   DATA[2489,28] := 261.6637;
   DATA[2489,29] := 12.11228;
   DATA[2489,30] := 1.723661;
   DATA[2489,31] := 1.271551;
   DATA[2489,32] := 0.7353967;
   DATA[2489,33] := 0.3084905;
   DATA[2489,34] := 2.0;
   DATA[2489,35] := 249.9199;
   DATA[2489,36] := 1.681991;
   DATA[2489,37] := 188.7817;
   DATA[2489,38] := 0.000128152;
   DATA[2489,39] := 1.0;
   DATA[2489,40] := 1.0;
   DATA[2490,0] := 2.585274;
   DATA[2490,1] := 868.7028;
   DATA[2490,2] := 2.0;
   DATA[2490,3] := 2.0;
   DATA[2490,4] := 262.3045;
   DATA[2490,5] := 8.396437;
   DATA[2490,6] := 329.7103;
   DATA[2490,7] := 2.455131;
   DATA[2490,8] := 2.0;
   DATA[2490,9] := 2.0;
   DATA[2490,10] := 2.0;
   DATA[2490,11] := 19.80601;
   DATA[2490,12] := 2.208884;
   DATA[2490,13] := 824.428;
   DATA[2490,14] := 1.0;
   DATA[2490,15] := 2.0;
   DATA[2490,16] := 1.0;
   DATA[2490,17] := 1.0;
   DATA[2490,18] := 1.0;
   DATA[2490,19] := 2.0;
   DATA[2490,20] := 148.808;
   DATA[2490,21] := 155.2166;
   DATA[2490,22] := 1.714798;
   DATA[2490,23] := 867.4699;
   DATA[2490,24] := 2.0;
   DATA[2490,25] := 2.0;
   DATA[2490,26] := 7.874135;
   DATA[2490,27] := 144.9628;
   DATA[2490,28] := 261.6637;
   DATA[2490,29] := 11.95847;
   DATA[2490,30] := 1.723661;
   DATA[2490,31] := 1.257333;
   DATA[2490,32] := 0.7353967;
   DATA[2490,33] := 0.3084905;
   DATA[2490,34] := 2.0;
   DATA[2490,35] := 249.9199;
   DATA[2490,36] := 1.681991;
   DATA[2490,37] := 188.7817;
   DATA[2490,38] := 0.000128152;
   DATA[2490,39] := 1.0;
   DATA[2490,40] := 1.0;
   DATA[2491,0] := 2.562854;
   DATA[2491,1] := 868.6635;
   DATA[2491,2] := 2.0;
   DATA[2491,3] := 2.0;
   DATA[2491,4] := 262.4007;
   DATA[2491,5] := 8.396437;
   DATA[2491,6] := 329.7103;
   DATA[2491,7] := 2.4559;
   DATA[2491,8] := 2.0;
   DATA[2491,9] := 2.0;
   DATA[2491,10] := 2.0;
   DATA[2491,11] := 19.77079;
   DATA[2491,12] := 2.208884;
   DATA[2491,13] := 825.0289;
   DATA[2491,14] := 1.0;
   DATA[2491,15] := 2.0;
   DATA[2491,16] := 1.0;
   DATA[2491,17] := 1.0;
   DATA[2491,18] := 1.0;
   DATA[2491,19] := 2.0;
   DATA[2491,20] := 148.808;
   DATA[2491,21] := 155.2166;
   DATA[2491,22] := 1.71608;
   DATA[2491,23] := 867.5468;
   DATA[2491,24] := 2.0;
   DATA[2491,25] := 2.0;
   DATA[2491,26] := 7.874135;
   DATA[2491,27] := 144.9628;
   DATA[2491,28] := 261.5355;
   DATA[2491,29] := 11.95847;
   DATA[2491,30] := 1.72507;
   DATA[2491,31] := 1.256565;
   DATA[2491,32] := 0.7353967;
   DATA[2491,33] := 0.3084905;
   DATA[2491,34] := 2.0;
   DATA[2491,35] := 249.9199;
   DATA[2491,36] := 1.681991;
   DATA[2491,37] := 188.7817;
   DATA[2491,38] := 0.000128152;
   DATA[2491,39] := 1.0;
   DATA[2491,40] := 1.0;
   DATA[2492,0] := 2.540115;
   DATA[2492,1] := 869.0953;
   DATA[2492,2] := 2.0;
   DATA[2492,3] := 2.0;
   DATA[2492,4] := 262.4007;
   DATA[2492,5] := 8.396437;
   DATA[2492,6] := 329.6591;
   DATA[2492,7] := 2.4559;
   DATA[2492,8] := 2.0;
   DATA[2492,9] := 2.0;
   DATA[2492,10] := 2.0;
   DATA[2492,11] := 19.72598;
   DATA[2492,12] := 2.208884;
   DATA[2492,13] := 825.0689;
   DATA[2492,14] := 1.0;
   DATA[2492,15] := 2.0;
   DATA[2492,16] := 1.0;
   DATA[2492,17] := 1.0;
   DATA[2492,18] := 1.0;
   DATA[2492,19] := 2.0;
   DATA[2492,20] := 148.808;
   DATA[2492,21] := 155.2166;
   DATA[2492,22] := 1.71608;
   DATA[2492,23] := 867.739;
   DATA[2492,24] := 2.0;
   DATA[2492,25] := 2.0;
   DATA[2492,26] := 7.874135;
   DATA[2492,27] := 144.9628;
   DATA[2492,28] := 261.5034;
   DATA[2492,29] := 11.95847;
   DATA[2492,30] := 1.72507;
   DATA[2492,31] := 1.261176;
   DATA[2492,32] := 0.7353967;
   DATA[2492,33] := 0.3084905;
   DATA[2492,34] := 2.0;
   DATA[2492,35] := 249.9199;
   DATA[2492,36] := 1.649953;
   DATA[2492,37] := 188.7817;
   DATA[2492,38] := 0.000128152;
   DATA[2492,39] := 1.0;
   DATA[2492,40] := 1.0;
   DATA[2493,0] := 2.524421;
   DATA[2493,1] := 868.7028;
   DATA[2493,2] := 2.0;
   DATA[2493,3] := 2.0;
   DATA[2493,4] := 262.4007;
   DATA[2493,5] := 8.395475;
   DATA[2493,6] := 329.6591;
   DATA[2493,7] := 2.4559;
   DATA[2493,8] := 2.0;
   DATA[2493,9] := 2.0;
   DATA[2493,10] := 2.0;
   DATA[2493,11] := 19.70357;
   DATA[2493,12] := 2.208884;
   DATA[2493,13] := 825.3493;
   DATA[2493,14] := 1.0;
   DATA[2493,15] := 2.0;
   DATA[2493,16] := 1.0;
   DATA[2493,17] := 1.0;
   DATA[2493,18] := 1.0;
   DATA[2493,19] := 2.0;
   DATA[2493,20] := 148.808;
   DATA[2493,21] := 155.2166;
   DATA[2493,22] := 1.71608;
   DATA[2493,23] := 867.6237;
   DATA[2493,24] := 2.0;
   DATA[2493,25] := 2.0;
   DATA[2493,26] := 7.874135;
   DATA[2493,27] := 144.8347;
   DATA[2493,28] := 261.5034;
   DATA[2493,29] := 11.95847;
   DATA[2493,30] := 1.725711;
   DATA[2493,31] := 1.271423;
   DATA[2493,32] := 0.7353967;
   DATA[2493,33] := 0.3084905;
   DATA[2493,34] := 2.0;
   DATA[2493,35] := 249.9199;
   DATA[2493,36] := 1.649953;
   DATA[2493,37] := 188.7817;
   DATA[2493,38] := 0.000128152;
   DATA[2493,39] := 1.0;
   DATA[2493,40] := 1.0;
   DATA[2494,0] := 2.510329;
   DATA[2494,1] := 868.7028;
   DATA[2494,2] := 2.0;
   DATA[2494,3] := 2.0;
   DATA[2494,4] := 262.4007;
   DATA[2494,5] := 8.393873;
   DATA[2494,6] := 329.454;
   DATA[2494,7] := 2.455003;
   DATA[2494,8] := 2.0;
   DATA[2494,9] := 2.0;
   DATA[2494,10] := 2.0;
   DATA[2494,11] := 19.67796;
   DATA[2494,12] := 2.208884;
   DATA[2494,13] := 825.7899;
   DATA[2494,14] := 1.0;
   DATA[2494,15] := 2.0;
   DATA[2494,16] := 1.0;
   DATA[2494,17] := 1.0;
   DATA[2494,18] := 1.0;
   DATA[2494,19] := 2.0;
   DATA[2494,20] := 148.808;
   DATA[2494,21] := 155.2166;
   DATA[2494,22] := 1.717746;
   DATA[2494,23] := 867.8159;
   DATA[2494,24] := 2.0;
   DATA[2494,25] := 2.0;
   DATA[2494,26] := 7.874135;
   DATA[2494,27] := 144.7065;
   DATA[2494,28] := 261.5034;
   DATA[2494,29] := 11.95847;
   DATA[2494,30] := 1.725711;
   DATA[2494,31] := 1.280902;
   DATA[2494,32] := 0.7353967;
   DATA[2494,33] := 0.3084905;
   DATA[2494,34] := 2.0;
   DATA[2494,35] := 249.9199;
   DATA[2494,36] := 1.649953;
   DATA[2494,37] := 188.8618;
   DATA[2494,38] := 0.000128152;
   DATA[2494,39] := 1.0;
   DATA[2494,40] := 1.0;
   DATA[2495,0] := 2.496877;
   DATA[2495,1] := 868.428;
   DATA[2495,2] := 2.0;
   DATA[2495,3] := 2.0;
   DATA[2495,4] := 262.4007;
   DATA[2495,5] := 8.393873;
   DATA[2495,6] := 329.454;
   DATA[2495,7] := 2.454362;
   DATA[2495,8] := 2.0;
   DATA[2495,9] := 2.0;
   DATA[2495,10] := 2.0;
   DATA[2495,11] := 19.65555;
   DATA[2495,12] := 2.208884;
   DATA[2495,13] := 825.87;
   DATA[2495,14] := 1.0;
   DATA[2495,15] := 2.0;
   DATA[2495,16] := 1.0;
   DATA[2495,17] := 1.0;
   DATA[2495,18] := 1.0;
   DATA[2495,19] := 2.0;
   DATA[2495,20] := 148.808;
   DATA[2495,21] := 155.2166;
   DATA[2495,22] := 1.717746;
   DATA[2495,23] := 868.1235;
   DATA[2495,24] := 2.0;
   DATA[2495,25] := 2.0;
   DATA[2495,26] := 7.874135;
   DATA[2495,27] := 144.7065;
   DATA[2495,28] := 261.5034;
   DATA[2495,29] := 11.95847;
   DATA[2495,30] := 1.725711;
   DATA[2495,31] := 1.291405;
   DATA[2495,32] := 0.7353967;
   DATA[2495,33] := 0.3084905;
   DATA[2495,34] := 2.0;
   DATA[2495,35] := 250.0;
   DATA[2495,36] := 1.649953;
   DATA[2495,37] := 188.8939;
   DATA[2495,38] := 0.000128152;
   DATA[2495,39] := 1.0;
   DATA[2495,40] := 1.0;
   DATA[2496,0] := 2.4767;
   DATA[2496,1] := 868.7421;
   DATA[2496,2] := 2.0;
   DATA[2496,3] := 2.0;
   DATA[2496,4] := 262.4007;
   DATA[2496,5] := 8.393873;
   DATA[2496,6] := 329.454;
   DATA[2496,7] := 2.454362;
   DATA[2496,8] := 2.0;
   DATA[2496,9] := 2.0;
   DATA[2496,10] := 2.0;
   DATA[2496,11] := 19.65555;
   DATA[2496,12] := 2.208244;
   DATA[2496,13] := 826.1504;
   DATA[2496,14] := 1.0;
   DATA[2496,15] := 2.0;
   DATA[2496,16] := 1.0;
   DATA[2496,17] := 1.0;
   DATA[2496,18] := 1.0;
   DATA[2496,19] := 2.0;
   DATA[2496,20] := 148.808;
   DATA[2496,21] := 155.2166;
   DATA[2496,22] := 1.717746;
   DATA[2496,23] := 867.8159;
   DATA[2496,24] := 2.0;
   DATA[2496,25] := 2.0;
   DATA[2496,26] := 7.874135;
   DATA[2496,27] := 144.7065;
   DATA[2496,28] := 261.5034;
   DATA[2496,29] := 11.95847;
   DATA[2496,30] := 1.725711;
   DATA[2496,31] := 1.287947;
   DATA[2496,32] := 0.7353967;
   DATA[2496,33] := 0.3084905;
   DATA[2496,34] := 2.0;
   DATA[2496,35] := 250.032;
   DATA[2496,36] := 1.778105;
   DATA[2496,37] := 188.8939;
   DATA[2496,38] := 0.000128152;
   DATA[2496,39] := 1.0;
   DATA[2496,40] := 1.0;
   DATA[2497,0] := 2.459405;
   DATA[2497,1] := 868.899;
   DATA[2497,2] := 2.0;
   DATA[2497,3] := 2.0;
   DATA[2497,4] := 262.4007;
   DATA[2497,5] := 8.393873;
   DATA[2497,6] := 329.454;
   DATA[2497,7] := 2.454362;
   DATA[2497,8] := 2.0;
   DATA[2497,9] := 2.0;
   DATA[2497,10] := 2.0;
   DATA[2497,11] := 19.65555;
   DATA[2497,12] := 2.208244;
   DATA[2497,13] := 826.5509;
   DATA[2497,14] := 1.0;
   DATA[2497,15] := 2.0;
   DATA[2497,16] := 1.0;
   DATA[2497,17] := 1.0;
   DATA[2497,18] := 1.0;
   DATA[2497,19] := 2.0;
   DATA[2497,20] := 148.808;
   DATA[2497,21] := 155.2935;
   DATA[2497,22] := 1.717746;
   DATA[2497,23] := 868.0466;
   DATA[2497,24] := 2.0;
   DATA[2497,25] := 2.0;
   DATA[2497,26] := 7.874135;
   DATA[2497,27] := 144.7065;
   DATA[2497,28] := 261.5034;
   DATA[2497,29] := 11.95847;
   DATA[2497,30] := 1.725711;
   DATA[2497,31] := 1.27834;
   DATA[2497,32] := 0.7353967;
   DATA[2497,33] := 0.3084905;
   DATA[2497,34] := 2.0;
   DATA[2497,35] := 250.032;
   DATA[2497,36] := 1.778105;
   DATA[2497,37] := 188.8939;
   DATA[2497,38] := 0.000128152;
   DATA[2497,39] := 1.0;
   DATA[2497,40] := 1.0;
   DATA[2498,0] := 2.44243;
   DATA[2498,1] := 868.9383;
   DATA[2498,2] := 2.0;
   DATA[2498,3] := 2.0;
   DATA[2498,4] := 262.1764;
   DATA[2498,5] := 8.393873;
   DATA[2498,6] := 329.454;
   DATA[2498,7] := 2.454362;
   DATA[2498,8] := 2.0;
   DATA[2498,9] := 2.0;
   DATA[2498,10] := 2.0;
   DATA[2498,11] := 19.65555;
   DATA[2498,12] := 2.208244;
   DATA[2498,13] := 826.3506;
   DATA[2498,14] := 1.0;
   DATA[2498,15] := 2.0;
   DATA[2498,16] := 1.0;
   DATA[2498,17] := 1.0;
   DATA[2498,18] := 1.0;
   DATA[2498,19] := 2.0;
   DATA[2498,20] := 148.808;
   DATA[2498,21] := 155.3448;
   DATA[2498,22] := 1.715439;
   DATA[2498,23] := 868.2004;
   DATA[2498,24] := 2.0;
   DATA[2498,25] := 2.0;
   DATA[2498,26] := 7.874135;
   DATA[2498,27] := 144.7065;
   DATA[2498,28] := 261.5034;
   DATA[2498,29] := 11.95847;
   DATA[2498,30] := 1.725711;
   DATA[2498,31] := 1.272064;
   DATA[2498,32] := 0.7353967;
   DATA[2498,33] := 0.3084905;
   DATA[2498,34] := 2.0;
   DATA[2498,35] := 250.032;
   DATA[2498,36] := 1.778105;
   DATA[2498,37] := 188.8939;
   DATA[2498,38] := 0.000128152;
   DATA[2498,39] := 1.0;
   DATA[2498,40] := 1.0;
   DATA[2499,0] := 2.429619;
   DATA[2499,1] := 869.0168;
   DATA[2499,2] := 2.0;
   DATA[2499,3] := 2.0;
   DATA[2499,4] := 262.1764;
   DATA[2499,5] := 8.396437;
   DATA[2499,6] := 329.454;
   DATA[2499,7] := 2.454362;
   DATA[2499,8] := 2.0;
   DATA[2499,9] := 2.0;
   DATA[2499,10] := 2.0;
   DATA[2499,11] := 19.65555;
   DATA[2499,12] := 2.207475;
   DATA[2499,13] := 826.2705;
   DATA[2499,14] := 1.0;
   DATA[2499,15] := 2.0;
   DATA[2499,16] := 1.0;
   DATA[2499,17] := 1.0;
   DATA[2499,18] := 1.0;
   DATA[2499,19] := 2.0;
   DATA[2499,20] := 148.808;
   DATA[2499,21] := 155.3448;
   DATA[2499,22] := 1.715439;
   DATA[2499,23] := 868.4312;
   DATA[2499,24] := 2.0;
   DATA[2499,25] := 2.0;
   DATA[2499,26] := 7.874135;
   DATA[2499,27] := 144.7065;
   DATA[2499,28] := 261.5034;
   DATA[2499,29] := 11.95847;
   DATA[2499,30] := 1.725711;
   DATA[2499,31] := 1.282951;
   DATA[2499,32] := 0.7353967;
   DATA[2499,33] := 0.3084905;
   DATA[2499,34] := 2.0;
   DATA[2499,35] := 250.032;
   DATA[2499,36] := 1.778105;
   DATA[2499,37] := 188.8939;
   DATA[2499,38] := 0.000128152;
   DATA[2499,39] := 1.0;
   DATA[2499,40] := 1.0;
   DATA[2500,0] := 2.428338;
   DATA[2500,1] := 868.9383;
   DATA[2500,2] := 2.0;
   DATA[2500,3] := 2.0;
   DATA[2500,4] := 262.1764;
   DATA[2500,5] := 8.396437;
   DATA[2500,6] := 329.5309;
   DATA[2500,7] := 2.4559;
   DATA[2500,8] := 2.0;
   DATA[2500,9] := 2.0;
   DATA[2500,10] := 2.0;
   DATA[2500,11] := 19.65555;
   DATA[2500,12] := 2.207475;
   DATA[2500,13] := 826.4307;
   DATA[2500,14] := 1.0;
   DATA[2500,15] := 2.0;
   DATA[2500,16] := 1.0;
   DATA[2500,17] := 1.0;
   DATA[2500,18] := 1.0;
   DATA[2500,19] := 2.0;
   DATA[2500,20] := 148.808;
   DATA[2500,21] := 155.3448;
   DATA[2500,22] := 1.716721;
   DATA[2500,23] := 868.3927;
   DATA[2500,24] := 2.0;
   DATA[2500,25] := 2.0;
   DATA[2500,26] := 7.874135;
   DATA[2500,27] := 144.7065;
   DATA[2500,28] := 261.5034;
   DATA[2500,29] := 11.95847;
   DATA[2500,30] := 1.725711;
   DATA[2500,31] := 1.301012;
   DATA[2500,32] := 0.7353967;
   DATA[2500,33] := 0.3084905;
   DATA[2500,34] := 2.0;
   DATA[2500,35] := 250.032;
   DATA[2500,36] := 1.778105;
   DATA[2500,37] := 188.8939;
   DATA[2500,38] := 0.000128152;
   DATA[2500,39] := 1.0;
   DATA[2500,40] := 1.0;
   DATA[2501,0] := 2.426416;
   DATA[2501,1] := 868.428;
   DATA[2501,2] := 2.0;
   DATA[2501,3] := 2.0;
   DATA[2501,4] := 262.1764;
   DATA[2501,5] := 8.396437;
   DATA[2501,6] := 329.5822;
   DATA[2501,7] := 2.456412;
   DATA[2501,8] := 2.0;
   DATA[2501,9] := 2.0;
   DATA[2501,10] := 2.0;
   DATA[2501,11] := 19.65555;
   DATA[2501,12] := 2.207475;
   DATA[2501,13] := 826.5909;
   DATA[2501,14] := 1.0;
   DATA[2501,15] := 2.0;
   DATA[2501,16] := 1.0;
   DATA[2501,17] := 1.0;
   DATA[2501,18] := 1.0;
   DATA[2501,19] := 2.0;
   DATA[2501,20] := 148.808;
   DATA[2501,21] := 155.3448;
   DATA[2501,22] := 1.71813;
   DATA[2501,23] := 868.5081;
   DATA[2501,24] := 2.0;
   DATA[2501,25] := 2.0;
   DATA[2501,26] := 7.874135;
   DATA[2501,27] := 144.7065;
   DATA[2501,28] := 261.5034;
   DATA[2501,29] := 11.95847;
   DATA[2501,30] := 1.725711;
   DATA[2501,31] := 1.311131;
   DATA[2501,32] := 0.7353967;
   DATA[2501,33] := 0.3084905;
   DATA[2501,34] := 2.0;
   DATA[2501,35] := 250.032;
   DATA[2501,36] := 1.69801;
   DATA[2501,37] := 188.8939;
   DATA[2501,38] := 0.000128152;
   DATA[2501,39] := 1.0;
   DATA[2501,40] := 1.0;
   DATA[2502,0] := 2.450758;
   DATA[2502,1] := 868.9383;
   DATA[2502,2] := 2.0;
   DATA[2502,3] := 2.0;
   DATA[2502,4] := 262.4007;
   DATA[2502,5] := 8.396437;
   DATA[2502,6] := 329.5822;
   DATA[2502,7] := 2.456412;
   DATA[2502,8] := 2.0;
   DATA[2502,9] := 2.0;
   DATA[2502,10] := 2.0;
   DATA[2502,11] := 19.65555;
   DATA[2502,12] := 2.207091;
   DATA[2502,13] := 826.4307;
   DATA[2502,14] := 1.0;
   DATA[2502,15] := 2.0;
   DATA[2502,16] := 1.0;
   DATA[2502,17] := 1.0;
   DATA[2502,18] := 1.0;
   DATA[2502,19] := 2.0;
   DATA[2502,20] := 148.808;
   DATA[2502,21] := 155.3448;
   DATA[2502,22] := 1.71813;
   DATA[2502,23] := 868.5465;
   DATA[2502,24] := 2.0;
   DATA[2502,25] := 2.0;
   DATA[2502,26] := 7.874135;
   DATA[2502,27] := 144.7065;
   DATA[2502,28] := 261.5034;
   DATA[2502,29] := 11.95847;
   DATA[2502,30] := 1.725583;
   DATA[2502,31] := 1.32125;
   DATA[2502,32] := 0.7353967;
   DATA[2502,33] := 0.3084905;
   DATA[2502,34] := 2.0;
   DATA[2502,35] := 250.032;
   DATA[2502,36] := 1.69801;
   DATA[2502,37] := 188.8939;
   DATA[2502,38] := 0.000128152;
   DATA[2502,39] := 1.0;
   DATA[2502,40] := 1.0;
   DATA[2503,0] := 2.504244;
   DATA[2503,1] := 868.8206;
   DATA[2503,2] := 2.0;
   DATA[2503,3] := 2.0;
   DATA[2503,4] := 262.4007;
   DATA[2503,5] := 8.396437;
   DATA[2503,6] := 329.5822;
   DATA[2503,7] := 2.456412;
   DATA[2503,8] := 2.0;
   DATA[2503,9] := 2.0;
   DATA[2503,10] := 2.0;
   DATA[2503,11] := 19.68756;
   DATA[2503,12] := 2.207091;
   DATA[2503,13] := 826.2305;
   DATA[2503,14] := 1.0;
   DATA[2503,15] := 2.0;
   DATA[2503,16] := 1.0;
   DATA[2503,17] := 1.0;
   DATA[2503,18] := 1.0;
   DATA[2503,19] := 2.0;
   DATA[2503,20] := 148.808;
   DATA[2503,21] := 155.3448;
   DATA[2503,22] := 1.71813;
   DATA[2503,23] := 868.6234;
   DATA[2503,24] := 2.0;
   DATA[2503,25] := 2.0;
   DATA[2503,26] := 7.874135;
   DATA[2503,27] := 144.7065;
   DATA[2503,28] := 261.5034;
   DATA[2503,29] := 11.95847;
   DATA[2503,30] := 1.725455;
   DATA[2503,31] := 1.322147;
   DATA[2503,32] := 0.7346286;
   DATA[2503,33] := 0.3084905;
   DATA[2503,34] := 2.0;
   DATA[2503,35] := 250.032;
   DATA[2503,36] := 1.69801;
   DATA[2503,37] := 188.8939;
   DATA[2503,38] := 0.000128152;
   DATA[2503,39] := 1.0;
   DATA[2503,40] := 1.0;
   DATA[2504,0] := 2.551965;
   DATA[2504,1] := 868.3495;
   DATA[2504,2] := 2.0;
   DATA[2504,3] := 2.0;
   DATA[2504,4] := 262.4007;
   DATA[2504,5] := 8.396437;
   DATA[2504,6] := 329.5822;
   DATA[2504,7] := 2.456412;
   DATA[2504,8] := 2.0;
   DATA[2504,9] := 2.0;
   DATA[2504,10] := 2.0;
   DATA[2504,11] := 19.68756;
   DATA[2504,12] := 2.207091;
   DATA[2504,13] := 826.0703;
   DATA[2504,14] := 1.0;
   DATA[2504,15] := 2.0;
   DATA[2504,16] := 1.0;
   DATA[2504,17] := 1.0;
   DATA[2504,18] := 1.0;
   DATA[2504,19] := 2.0;
   DATA[2504,20] := 148.808;
   DATA[2504,21] := 155.3448;
   DATA[2504,22] := 1.716849;
   DATA[2504,23] := 868.585;
   DATA[2504,24] := 2.0;
   DATA[2504,25] := 2.0;
   DATA[2504,26] := 7.874135;
   DATA[2504,27] := 144.7065;
   DATA[2504,28] := 261.5034;
   DATA[2504,29] := 11.95847;
   DATA[2504,30] := 1.72443;
   DATA[2504,31] := 1.315486;
   DATA[2504,32] := 0.7346286;
   DATA[2504,33] := 0.3084905;
   DATA[2504,34] := 2.0;
   DATA[2504,35] := 250.032;
   DATA[2504,36] := 1.69801;
   DATA[2504,37] := 188.8939;
   DATA[2504,38] := 0.000128152;
   DATA[2504,39] := 1.0;
   DATA[2504,40] := 1.0;
   DATA[2505,0] := 2.589117;
   DATA[2505,1] := 868.3102;
   DATA[2505,2] := 2.0;
   DATA[2505,3] := 2.0;
   DATA[2505,4] := 262.4007;
   DATA[2505,5] := 8.394514;
   DATA[2505,6] := 329.5822;
   DATA[2505,7] := 2.456412;
   DATA[2505,8] := 2.0;
   DATA[2505,9] := 2.0;
   DATA[2505,10] := 2.0;
   DATA[2505,11] := 19.61393;
   DATA[2505,12] := 2.207091;
   DATA[2505,13] := 826.1504;
   DATA[2505,14] := 1.0;
   DATA[2505,15] := 2.0;
   DATA[2505,16] := 1.0;
   DATA[2505,17] := 1.0;
   DATA[2505,18] := 1.0;
   DATA[2505,19] := 2.0;
   DATA[2505,20] := 148.808;
   DATA[2505,21] := 155.4473;
   DATA[2505,22] := 1.715183;
   DATA[2505,23] := 868.3542;
   DATA[2505,24] := 2.0;
   DATA[2505,25] := 2.0;
   DATA[2505,26] := 7.874135;
   DATA[2505,27] := 144.7065;
   DATA[2505,28] := 261.6637;
   DATA[2505,29] := 11.95847;
   DATA[2505,30] := 1.72443;
   DATA[2505,31] := 1.294992;
   DATA[2505,32] := 0.7346286;
   DATA[2505,33] := 0.3084905;
   DATA[2505,34] := 2.0;
   DATA[2505,35] := 250.032;
   DATA[2505,36] := 1.69801;
   DATA[2505,37] := 188.8779;
   DATA[2505,38] := 0.000128152;
   DATA[2505,39] := 1.0;
   DATA[2505,40] := 1.0;
   DATA[2506,0] := 2.621785;
   DATA[2506,1] := 868.2318;
   DATA[2506,2] := 2.0;
   DATA[2506,3] := 2.0;
   DATA[2506,4] := 262.4007;
   DATA[2506,5] := 8.394514;
   DATA[2506,6] := 329.5822;
   DATA[2506,7] := 2.456412;
   DATA[2506,8] := 2.0;
   DATA[2506,9] := 2.0;
   DATA[2506,10] := 2.0;
   DATA[2506,11] := 19.61393;
   DATA[2506,12] := 2.207091;
   DATA[2506,13] := 826.0302;
   DATA[2506,14] := 1.0;
   DATA[2506,15] := 2.0;
   DATA[2506,16] := 1.0;
   DATA[2506,17] := 1.0;
   DATA[2506,18] := 1.0;
   DATA[2506,19] := 2.0;
   DATA[2506,20] := 148.808;
   DATA[2506,21] := 155.4473;
   DATA[2506,22] := 1.715183;
   DATA[2506,23] := 868.7772;
   DATA[2506,24] := 2.0;
   DATA[2506,25] := 2.0;
   DATA[2506,26] := 7.874135;
   DATA[2506,27] := 144.7065;
   DATA[2506,28] := 261.6637;
   DATA[2506,29] := 11.95847;
   DATA[2506,30] := 1.72443;
   DATA[2506,31] := 1.275266;
   DATA[2506,32] := 0.7352687;
   DATA[2506,33] := 0.3084905;
   DATA[2506,34] := 2.0;
   DATA[2506,35] := 250.032;
   DATA[2506,36] := 1.69801;
   DATA[2506,37] := 188.8458;
   DATA[2506,38] := 0.000128152;
   DATA[2506,39] := 1.0;
   DATA[2506,40] := 1.0;
   DATA[2507,0] := 2.63844;
   DATA[2507,1] := 868.3102;
   DATA[2507,2] := 2.0;
   DATA[2507,3] := 2.0;
   DATA[2507,4] := 262.4007;
   DATA[2507,5] := 8.394514;
   DATA[2507,6] := 329.5822;
   DATA[2507,7] := 2.456412;
   DATA[2507,8] := 2.0;
   DATA[2507,9] := 2.0;
   DATA[2507,10] := 2.0;
   DATA[2507,11] := 19.66835;
   DATA[2507,12] := 2.207091;
   DATA[2507,13] := 825.9902;
   DATA[2507,14] := 1.0;
   DATA[2507,15] := 2.0;
   DATA[2507,16] := 1.0;
   DATA[2507,17] := 1.0;
   DATA[2507,18] := 1.0;
   DATA[2507,19] := 2.0;
   DATA[2507,20] := 148.808;
   DATA[2507,21] := 155.4473;
   DATA[2507,22] := 1.715183;
   DATA[2507,23] := 868.8157;
   DATA[2507,24] := 2.0;
   DATA[2507,25] := 2.0;
   DATA[2507,26] := 7.874135;
   DATA[2507,27] := 144.7065;
   DATA[2507,28] := 261.6637;
   DATA[2507,29] := 11.95847;
   DATA[2507,30] := 1.726865;
   DATA[2507,31] := 1.271551;
   DATA[2507,32] := 0.7352687;
   DATA[2507,33] := 0.3084905;
   DATA[2507,34] := 2.0;
   DATA[2507,35] := 250.032;
   DATA[2507,36] := 1.69801;
   DATA[2507,37] := 188.8458;
   DATA[2507,38] := 0.000128152;
   DATA[2507,39] := 1.0;
   DATA[2507,40] := 1.0;
   DATA[2508,0] := 2.652211;
   DATA[2508,1] := 867.6429;
   DATA[2508,2] := 2.0;
   DATA[2508,3] := 2.0;
   DATA[2508,4] := 262.4007;
   DATA[2508,5] := 8.394514;
   DATA[2508,6] := 329.5822;
   DATA[2508,7] := 2.456284;
   DATA[2508,8] := 2.0;
   DATA[2508,9] := 2.0;
   DATA[2508,10] := 2.0;
   DATA[2508,11] := 19.71957;
   DATA[2508,12] := 2.207091;
   DATA[2508,13] := 825.5896;
   DATA[2508,14] := 1.0;
   DATA[2508,15] := 2.0;
   DATA[2508,16] := 1.0;
   DATA[2508,17] := 1.0;
   DATA[2508,18] := 1.0;
   DATA[2508,19] := 2.0;
   DATA[2508,20] := 148.808;
   DATA[2508,21] := 155.4473;
   DATA[2508,22] := 1.715183;
   DATA[2508,23] := 868.7388;
   DATA[2508,24] := 2.0;
   DATA[2508,25] := 2.0;
   DATA[2508,26] := 7.874135;
   DATA[2508,27] := 144.7065;
   DATA[2508,28] := 261.6637;
   DATA[2508,29] := 11.95847;
   DATA[2508,30] := 1.726865;
   DATA[2508,31] := 1.261944;
   DATA[2508,32] := 0.7352687;
   DATA[2508,33] := 0.3084905;
   DATA[2508,34] := 2.0;
   DATA[2508,35] := 250.032;
   DATA[2508,36] := 1.69801;
   DATA[2508,37] := 188.8458;
   DATA[2508,38] := 0.000128152;
   DATA[2508,39] := 1.0;
   DATA[2508,40] := 1.0;
   DATA[2509,0] := 2.652211;
   DATA[2509,1] := 867.7215;
   DATA[2509,2] := 2.0;
   DATA[2509,3] := 2.0;
   DATA[2509,4] := 262.4007;
   DATA[2509,5] := 8.394514;
   DATA[2509,6] := 329.5822;
   DATA[2509,7] := 2.456284;
   DATA[2509,8] := 2.0;
   DATA[2509,9] := 2.0;
   DATA[2509,10] := 2.0;
   DATA[2509,11] := 19.74838;
   DATA[2509,12] := 2.207091;
   DATA[2509,13] := 825.3893;
   DATA[2509,14] := 1.0;
   DATA[2509,15] := 2.0;
   DATA[2509,16] := 1.0;
   DATA[2509,17] := 1.0;
   DATA[2509,18] := 1.0;
   DATA[2509,19] := 2.0;
   DATA[2509,20] := 148.808;
   DATA[2509,21] := 155.4473;
   DATA[2509,22] := 1.715183;
   DATA[2509,23] := 868.8926;
   DATA[2509,24] := 2.0;
   DATA[2509,25] := 2.0;
   DATA[2509,26] := 7.874135;
   DATA[2509,27] := 144.7065;
   DATA[2509,28] := 261.6637;
   DATA[2509,29] := 11.95847;
   DATA[2509,30] := 1.726865;
   DATA[2509,31] := 1.268861;
   DATA[2509,32] := 0.7352687;
   DATA[2509,33] := 0.3084905;
   DATA[2509,34] := 2.0;
   DATA[2509,35] := 250.032;
   DATA[2509,36] := 1.69801;
   DATA[2509,37] := 188.8458;
   DATA[2509,38] := 0.000128152;
   DATA[2509,39] := 1.0;
   DATA[2509,40] := 1.0;
   DATA[2510,0] := 2.628191;
   DATA[2510,1] := 867.5645;
   DATA[2510,2] := 2.0;
   DATA[2510,3] := 2.0;
   DATA[2510,4] := 262.4007;
   DATA[2510,5] := 8.394514;
   DATA[2510,6] := 329.5822;
   DATA[2510,7] := 2.456284;
   DATA[2510,8] := 2.0;
   DATA[2510,9] := 2.0;
   DATA[2510,10] := 2.0;
   DATA[2510,11] := 19.74838;
   DATA[2510,12] := 2.207091;
   DATA[2510,13] := 825.3493;
   DATA[2510,14] := 1.0;
   DATA[2510,15] := 2.0;
   DATA[2510,16] := 1.0;
   DATA[2510,17] := 1.0;
   DATA[2510,18] := 1.0;
   DATA[2510,19] := 2.0;
   DATA[2510,20] := 148.808;
   DATA[2510,21] := 155.4473;
   DATA[2510,22] := 1.715824;
   DATA[2510,23] := 869.2002;
   DATA[2510,24] := 2.0;
   DATA[2510,25] := 2.0;
   DATA[2510,26] := 7.874135;
   DATA[2510,27] := 144.7065;
   DATA[2510,28] := 261.6637;
   DATA[2510,29] := 11.95847;
   DATA[2510,30] := 1.726865;
   DATA[2510,31] := 1.271935;
   DATA[2510,32] := 0.7352687;
   DATA[2510,33] := 0.3084905;
   DATA[2510,34] := 2.0;
   DATA[2510,35] := 250.0641;
   DATA[2510,36] := 1.69801;
   DATA[2510,37] := 188.8618;
   DATA[2510,38] := 0.000128152;
   DATA[2510,39] := 1.0;
   DATA[2510,40] := 1.0;
   DATA[2511,0] := 2.613778;
   DATA[2511,1] := 867.1719;
   DATA[2511,2] := 2.0;
   DATA[2511,3] := 2.0;
   DATA[2511,4] := 262.4007;
   DATA[2511,5] := 8.394514;
   DATA[2511,6] := 329.5822;
   DATA[2511,7] := 2.456284;
   DATA[2511,8] := 2.0;
   DATA[2511,9] := 2.0;
   DATA[2511,10] := 2.0;
   DATA[2511,11] := 19.74838;
   DATA[2511,12] := 2.207091;
   DATA[2511,13] := 825.1891;
   DATA[2511,14] := 1.0;
   DATA[2511,15] := 2.0;
   DATA[2511,16] := 1.0;
   DATA[2511,17] := 1.0;
   DATA[2511,18] := 1.0;
   DATA[2511,19] := 2.0;
   DATA[2511,20] := 148.808;
   DATA[2511,21] := 155.4473;
   DATA[2511,22] := 1.717361;
   DATA[2511,23] := 869.3925;
   DATA[2511,24] := 2.0;
   DATA[2511,25] := 2.0;
   DATA[2511,26] := 7.874135;
   DATA[2511,27] := 144.7834;
   DATA[2511,28] := 261.6637;
   DATA[2511,29] := 12.26609;
   DATA[2511,30] := 1.726865;
   DATA[2511,31] := 1.265531;
   DATA[2511,32] := 0.7352687;
   DATA[2511,33] := 0.3084905;
   DATA[2511,34] := 2.0;
   DATA[2511,35] := 250.1923;
   DATA[2511,36] := 1.69801;
   DATA[2511,37] := 189.006;
   DATA[2511,38] := 0.000128152;
   DATA[2511,39] := 1.0;
   DATA[2511,40] := 1.0;
   DATA[2512,0] := 2.607373;
   DATA[2512,1] := 866.7794;
   DATA[2512,2] := 2.0;
   DATA[2512,3] := 2.0;
   DATA[2512,4] := 262.4007;
   DATA[2512,5] := 8.394514;
   DATA[2512,6] := 329.5822;
   DATA[2512,7] := 2.456284;
   DATA[2512,8] := 2.0;
   DATA[2512,9] := 2.0;
   DATA[2512,10] := 2.0;
   DATA[2512,11] := 19.74838;
   DATA[2512,12] := 2.207091;
   DATA[2512,13] := 825.2291;
   DATA[2512,14] := 1.0;
   DATA[2512,15] := 2.0;
   DATA[2512,16] := 1.0;
   DATA[2512,17] := 1.0;
   DATA[2512,18] := 1.0;
   DATA[2512,19] := 2.0;
   DATA[2512,20] := 148.808;
   DATA[2512,21] := 155.4473;
   DATA[2512,22] := 1.718387;
   DATA[2512,23] := 869.3925;
   DATA[2512,24] := 2.0;
   DATA[2512,25] := 2.0;
   DATA[2512,26] := 7.874135;
   DATA[2512,27] := 144.7834;
   DATA[2512,28] := 261.6637;
   DATA[2512,29] := 12.26609;
   DATA[2512,30] := 1.726865;
   DATA[2512,31] := 1.26963;
   DATA[2512,32] := 0.7352687;
   DATA[2512,33] := 0.3084905;
   DATA[2512,34] := 2.0;
   DATA[2512,35] := 250.1923;
   DATA[2512,36] := 1.69801;
   DATA[2512,37] := 189.006;
   DATA[2512,38] := 0.000128152;
   DATA[2512,39] := 1.0;
   DATA[2512,40] := 1.0;
   DATA[2513,0] := 2.601608;
   DATA[2513,1] := 866.7402;
   DATA[2513,2] := 2.0;
   DATA[2513,3] := 2.0;
   DATA[2513,4] := 262.4007;
   DATA[2513,5] := 8.394514;
   DATA[2513,6] := 329.5822;
   DATA[2513,7] := 2.456284;
   DATA[2513,8] := 2.0;
   DATA[2513,9] := 2.0;
   DATA[2513,10] := 2.0;
   DATA[2513,11] := 19.73878;
   DATA[2513,12] := 2.207091;
   DATA[2513,13] := 825.0289;
   DATA[2513,14] := 1.0;
   DATA[2513,15] := 2.0;
   DATA[2513,16] := 1.0;
   DATA[2513,17] := 1.0;
   DATA[2513,18] := 1.0;
   DATA[2513,19] := 2.0;
   DATA[2513,20] := 148.808;
   DATA[2513,21] := 155.4473;
   DATA[2513,22] := 1.718643;
   DATA[2513,23] := 869.3925;
   DATA[2513,24] := 2.0;
   DATA[2513,25] := 2.0;
   DATA[2513,26] := 7.874135;
   DATA[2513,27] := 144.7834;
   DATA[2513,28] := 261.6637;
   DATA[2513,29] := 12.15073;
   DATA[2513,30] := 1.726609;
   DATA[2513,31] := 1.28372;
   DATA[2513,32] := 0.7352687;
   DATA[2513,33] := 0.3084905;
   DATA[2513,34] := 2.0;
   DATA[2513,35] := 250.1923;
   DATA[2513,36] := 1.69801;
   DATA[2513,37] := 189.006;
   DATA[2513,38] := 0.000128152;
   DATA[2513,39] := 1.0;
   DATA[2513,40] := 1.0;
   DATA[2514,0] := 2.586555;
   DATA[2514,1] := 867.0542;
   DATA[2514,2] := 2.0;
   DATA[2514,3] := 2.0;
   DATA[2514,4] := 262.4007;
   DATA[2514,5] := 8.394514;
   DATA[2514,6] := 329.5822;
   DATA[2514,7] := 2.456284;
   DATA[2514,8] := 2.0;
   DATA[2514,9] := 2.0;
   DATA[2514,10] := 2.0;
   DATA[2514,11] := 19.73878;
   DATA[2514,12] := 2.207091;
   DATA[2514,13] := 824.8286;
   DATA[2514,14] := 1.0;
   DATA[2514,15] := 2.0;
   DATA[2514,16] := 1.0;
   DATA[2514,17] := 1.0;
   DATA[2514,18] := 1.0;
   DATA[2514,19] := 2.0;
   DATA[2514,20] := 148.808;
   DATA[2514,21] := 155.4473;
   DATA[2514,22] := 1.718643;
   DATA[2514,23] := 869.9308;
   DATA[2514,24] := 2.0;
   DATA[2514,25] := 2.0;
   DATA[2514,26] := 7.874135;
   DATA[2514,27] := 144.7834;
   DATA[2514,28] := 261.6637;
   DATA[2514,29] := 12.15073;
   DATA[2514,30] := 1.72507;
   DATA[2514,31] := 1.291533;
   DATA[2514,32] := 0.7352687;
   DATA[2514,33] := 0.3084905;
   DATA[2514,34] := 2.0;
   DATA[2514,35] := 250.1923;
   DATA[2514,36] := 1.69801;
   DATA[2514,37] := 189.006;
   DATA[2514,38] := 0.000128152;
   DATA[2514,39] := 1.0;
   DATA[2514,40] := 1.0;
   DATA[2515,0] := 2.572142;
   DATA[2515,1] := 867.3682;
   DATA[2515,2] := 2.0;
   DATA[2515,3] := 2.0;
   DATA[2515,4] := 262.4007;
   DATA[2515,5] := 8.394514;
   DATA[2515,6] := 329.5822;
   DATA[2515,7] := 2.456284;
   DATA[2515,8] := 2.0;
   DATA[2515,9] := 2.0;
   DATA[2515,10] := 2.0;
   DATA[2515,11] := 19.81561;
   DATA[2515,12] := 2.207091;
   DATA[2515,13] := 824.5883;
   DATA[2515,14] := 1.0;
   DATA[2515,15] := 2.0;
   DATA[2515,16] := 1.0;
   DATA[2515,17] := 1.0;
   DATA[2515,18] := 1.0;
   DATA[2515,19] := 2.0;
   DATA[2515,20] := 148.808;
   DATA[2515,21] := 155.4473;
   DATA[2515,22] := 1.718643;
   DATA[2515,23] := 870.0077;
   DATA[2515,24] := 2.0;
   DATA[2515,25] := 2.0;
   DATA[2515,26] := 7.874135;
   DATA[2515,27] := 144.7834;
   DATA[2515,28] := 261.6637;
   DATA[2515,29] := 12.15073;
   DATA[2515,30] := 1.72507;
   DATA[2515,31] := 1.291533;
   DATA[2515,32] := 0.7352687;
   DATA[2515,33] := 0.3084905;
   DATA[2515,34] := 2.0;
   DATA[2515,35] := 250.1923;
   DATA[2515,36] := 1.69801;
   DATA[2515,37] := 189.006;
   DATA[2515,38] := 0.000128152;
   DATA[2515,39] := 1.0;
   DATA[2515,40] := 1.0;
   DATA[2516,0] := 2.555168;
   DATA[2516,1] := 867.8392;
   DATA[2516,2] := 2.0;
   DATA[2516,3] := 2.0;
   DATA[2516,4] := 262.4007;
   DATA[2516,5] := 8.395155;
   DATA[2516,6] := 329.5822;
   DATA[2516,7] := 2.456284;
   DATA[2516,8] := 2.0;
   DATA[2516,9] := 2.0;
   DATA[2516,10] := 2.0;
   DATA[2516,11] := 19.81561;
   DATA[2516,12] := 2.209013;
   DATA[2516,13] := 824.9888;
   DATA[2516,14] := 1.0;
   DATA[2516,15] := 2.0;
   DATA[2516,16] := 1.0;
   DATA[2516,17] := 1.0;
   DATA[2516,18] := 1.0;
   DATA[2516,19] := 2.0;
   DATA[2516,20] := 148.808;
   DATA[2516,21] := 155.4473;
   DATA[2516,22] := 1.717874;
   DATA[2516,23] := 869.8923;
   DATA[2516,24] := 2.0;
   DATA[2516,25] := 2.0;
   DATA[2516,26] := 7.874135;
   DATA[2516,27] := 144.7834;
   DATA[2516,28] := 261.6637;
   DATA[2516,29] := 11.88157;
   DATA[2516,30] := 1.72507;
   DATA[2516,31] := 1.291533;
   DATA[2516,32] := 0.7352687;
   DATA[2516,33] := 0.3084905;
   DATA[2516,34] := 2.0;
   DATA[2516,35] := 250.1923;
   DATA[2516,36] := 1.69801;
   DATA[2516,37] := 189.006;
   DATA[2516,38] := 0.000128152;
   DATA[2516,39] := 1.0;
   DATA[2516,40] := 1.0;
   DATA[2517,0] := 2.541075;
   DATA[2517,1] := 867.8785;
   DATA[2517,2] := 2.0;
   DATA[2517,3] := 2.0;
   DATA[2517,4] := 262.3366;
   DATA[2517,5] := 8.396757;
   DATA[2517,6] := 329.5822;
   DATA[2517,7] := 2.455131;
   DATA[2517,8] := 2.0;
   DATA[2517,9] := 2.0;
   DATA[2517,10] := 2.0;
   DATA[2517,11] := 19.81561;
   DATA[2517,12] := 2.209013;
   DATA[2517,13] := 825.1891;
   DATA[2517,14] := 1.0;
   DATA[2517,15] := 2.0;
   DATA[2517,16] := 1.0;
   DATA[2517,17] := 1.0;
   DATA[2517,18] := 1.0;
   DATA[2517,19] := 2.0;
   DATA[2517,20] := 148.808;
   DATA[2517,21] := 155.4473;
   DATA[2517,22] := 1.717489;
   DATA[2517,23] := 870.2;
   DATA[2517,24] := 2.0;
   DATA[2517,25] := 2.0;
   DATA[2517,26] := 7.874135;
   DATA[2517,27] := 144.7834;
   DATA[2517,28] := 261.6637;
   DATA[2517,29] := 11.88157;
   DATA[2517,30] := 1.72507;
   DATA[2517,31] := 1.282823;
   DATA[2517,32] := 0.7352687;
   DATA[2517,33] := 0.3084905;
   DATA[2517,34] := 2.0;
   DATA[2517,35] := 250.0961;
   DATA[2517,36] := 1.69801;
   DATA[2517,37] := 189.006;
   DATA[2517,38] := 0.000128152;
   DATA[2517,39] := 1.0;
   DATA[2517,40] := 1.0;
   DATA[2518,0] := 2.521218;
   DATA[2518,1] := 867.6822;
   DATA[2518,2] := 2.0;
   DATA[2518,3] := 2.0;
   DATA[2518,4] := 262.3366;
   DATA[2518,5] := 8.396757;
   DATA[2518,6] := 329.5822;
   DATA[2518,7] := 2.453209;
   DATA[2518,8] := 2.0;
   DATA[2518,9] := 2.0;
   DATA[2518,10] := 2.0;
   DATA[2518,11] := 19.69076;
   DATA[2518,12] := 2.209013;
   DATA[2518,13] := 825.87;
   DATA[2518,14] := 1.0;
   DATA[2518,15] := 2.0;
   DATA[2518,16] := 1.0;
   DATA[2518,17] := 1.0;
   DATA[2518,18] := 1.0;
   DATA[2518,19] := 2.0;
   DATA[2518,20] := 148.808;
   DATA[2518,21] := 155.4473;
   DATA[2518,22] := 1.717361;
   DATA[2518,23] := 869.9692;
   DATA[2518,24] := 2.0;
   DATA[2518,25] := 2.0;
   DATA[2518,26] := 7.874135;
   DATA[2518,27] := 144.527;
   DATA[2518,28] := 261.6637;
   DATA[2518,29] := 11.88157;
   DATA[2518,30] := 1.72507;
   DATA[2518,31] := 1.281798;
   DATA[2518,32] := 0.7352687;
   DATA[2518,33] := 0.3084905;
   DATA[2518,34] := 2.0;
   DATA[2518,35] := 250.032;
   DATA[2518,36] := 1.617916;
   DATA[2518,37] := 188.9259;
   DATA[2518,38] := 0.000128152;
   DATA[2518,39] := 1.0;
   DATA[2518,40] := 1.0;
   DATA[2519,0] := 2.509688;
   DATA[2519,1] := 867.7607;
   DATA[2519,2] := 2.0;
   DATA[2519,3] := 2.0;
   DATA[2519,4] := 262.3366;
   DATA[2519,5] := 8.396757;
   DATA[2519,6] := 329.5822;
   DATA[2519,7] := 2.453209;
   DATA[2519,8] := 2.0;
   DATA[2519,9] := 2.0;
   DATA[2519,10] := 2.0;
   DATA[2519,11] := 19.65875;
   DATA[2519,12] := 2.209013;
   DATA[2519,13] := 825.9501;
   DATA[2519,14] := 1.0;
   DATA[2519,15] := 2.0;
   DATA[2519,16] := 1.0;
   DATA[2519,17] := 1.0;
   DATA[2519,18] := 1.0;
   DATA[2519,19] := 2.0;
   DATA[2519,20] := 148.808;
   DATA[2519,21] := 155.4473;
   DATA[2519,22] := 1.717361;
   DATA[2519,23] := 870.3153;
   DATA[2519,24] := 2.0;
   DATA[2519,25] := 2.0;
   DATA[2519,26] := 7.874135;
   DATA[2519,27] := 144.527;
   DATA[2519,28] := 261.6637;
   DATA[2519,29] := 11.88157;
   DATA[2519,30] := 1.72507;
   DATA[2519,31] := 1.29307;
   DATA[2519,32] := 0.7352687;
   DATA[2519,33] := 0.3084905;
   DATA[2519,34] := 2.0;
   DATA[2519,35] := 250.032;
   DATA[2519,36] := 1.617916;
   DATA[2519,37] := 188.8618;
   DATA[2519,38] := 0.000128152;
   DATA[2519,39] := 1.0;
   DATA[2519,40] := 1.0;
   DATA[2520,0] := 2.491112;
   DATA[2520,1] := 867.957;
   DATA[2520,2] := 2.0;
   DATA[2520,3] := 2.0;
   DATA[2520,4] := 262.3366;
   DATA[2520,5] := 8.39868;
   DATA[2520,6] := 329.5822;
   DATA[2520,7] := 2.45308;
   DATA[2520,8] := 2.0;
   DATA[2520,9] := 2.0;
   DATA[2520,10] := 2.0;
   DATA[2520,11] := 19.65875;
   DATA[2520,12] := 2.209013;
   DATA[2520,13] := 826.2305;
   DATA[2520,14] := 1.0;
   DATA[2520,15] := 2.0;
   DATA[2520,16] := 1.0;
   DATA[2520,17] := 1.0;
   DATA[2520,18] := 1.0;
   DATA[2520,19] := 2.0;
   DATA[2520,20] := 148.808;
   DATA[2520,21] := 155.4473;
   DATA[2520,22] := 1.717361;
   DATA[2520,23] := 870.5076;
   DATA[2520,24] := 2.0;
   DATA[2520,25] := 2.0;
   DATA[2520,26] := 7.874135;
   DATA[2520,27] := 144.527;
   DATA[2520,28] := 261.5355;
   DATA[2520,29] := 11.88157;
   DATA[2520,30] := 1.72507;
   DATA[2520,31] := 1.302037;
   DATA[2520,32] := 0.7352687;
   DATA[2520,33] := 0.3084905;
   DATA[2520,34] := 2.0;
   DATA[2520,35] := 250.032;
   DATA[2520,36] := 1.617916;
   DATA[2520,37] := 188.8618;
   DATA[2520,38] := 0.000128152;
   DATA[2520,39] := 1.0;
   DATA[2520,40] := 1.0;
   DATA[2521,0] := 2.480223;
   DATA[2521,1] := 868.1533;
   DATA[2521,2] := 2.0;
   DATA[2521,3] := 2.0;
   DATA[2521,4] := 262.3366;
   DATA[2521,5] := 8.399961;
   DATA[2521,6] := 329.5822;
   DATA[2521,7] := 2.452055;
   DATA[2521,8] := 2.0;
   DATA[2521,9] := 2.0;
   DATA[2521,10] := 2.0;
   DATA[2521,11] := 19.65875;
   DATA[2521,12] := 2.209013;
   DATA[2521,13] := 826.3907;
   DATA[2521,14] := 1.0;
   DATA[2521,15] := 2.0;
   DATA[2521,16] := 1.0;
   DATA[2521,17] := 1.0;
   DATA[2521,18] := 1.0;
   DATA[2521,19] := 2.0;
   DATA[2521,20] := 148.808;
   DATA[2521,21] := 155.4473;
   DATA[2521,22] := 1.716208;
   DATA[2521,23] := 870.4691;
   DATA[2521,24] := 2.0;
   DATA[2521,25] := 2.0;
   DATA[2521,26] := 7.874135;
   DATA[2521,27] := 144.527;
   DATA[2521,28] := 261.5355;
   DATA[2521,29] := 12.03538;
   DATA[2521,30] := 1.72507;
   DATA[2521,31] := 1.302037;
   DATA[2521,32] := 0.7352687;
   DATA[2521,33] := 0.3084905;
   DATA[2521,34] := 2.0;
   DATA[2521,35] := 250.032;
   DATA[2521,36] := 1.730048;
   DATA[2521,37] := 188.8618;
   DATA[2521,38] := 0.000128152;
   DATA[2521,39] := 1.0;
   DATA[2521,40] := 1.0;
   DATA[2522,0] := 2.462287;
   DATA[2522,1] := 868.3102;
   DATA[2522,2] := 2.0;
   DATA[2522,3] := 2.0;
   DATA[2522,4] := 262.3366;
   DATA[2522,5] := 8.399961;
   DATA[2522,6] := 329.5822;
   DATA[2522,7] := 2.451671;
   DATA[2522,8] := 2.0;
   DATA[2522,9] := 2.0;
   DATA[2522,10] := 2.0;
   DATA[2522,11] := 19.65875;
   DATA[2522,12] := 2.208244;
   DATA[2522,13] := 826.4708;
   DATA[2522,14] := 1.0;
   DATA[2522,15] := 2.0;
   DATA[2522,16] := 1.0;
   DATA[2522,17] := 1.0;
   DATA[2522,18] := 1.0;
   DATA[2522,19] := 2.0;
   DATA[2522,20] := 148.808;
   DATA[2522,21] := 155.4473;
   DATA[2522,22] := 1.716208;
   DATA[2522,23] := 870.5845;
   DATA[2522,24] := 2.0;
   DATA[2522,25] := 2.0;
   DATA[2522,26] := 7.874135;
   DATA[2522,27] := 144.527;
   DATA[2522,28] := 261.5355;
   DATA[2522,29] := 12.03538;
   DATA[2522,30] := 1.72507;
   DATA[2522,31] := 1.302037;
   DATA[2522,32] := 0.7352687;
   DATA[2522,33] := 0.3084905;
   DATA[2522,34] := 2.0;
   DATA[2522,35] := 250.032;
   DATA[2522,36] := 1.730048;
   DATA[2522,37] := 188.8618;
   DATA[2522,38] := 0.000128152;
   DATA[2522,39] := 1.0;
   DATA[2522,40] := 1.0;
   DATA[2523,0] := 2.447555;
   DATA[2523,1] := 868.1533;
   DATA[2523,2] := 2.0;
   DATA[2523,3] := 2.0;
   DATA[2523,4] := 262.3366;
   DATA[2523,5] := 8.399961;
   DATA[2523,6] := 329.5822;
   DATA[2523,7] := 2.451671;
   DATA[2523,8] := 2.0;
   DATA[2523,9] := 2.0;
   DATA[2523,10] := 2.0;
   DATA[2523,11] := 19.65875;
   DATA[2523,12] := 2.208116;
   DATA[2523,13] := 826.3907;
   DATA[2523,14] := 1.0;
   DATA[2523,15] := 2.0;
   DATA[2523,16] := 1.0;
   DATA[2523,17] := 1.0;
   DATA[2523,18] := 1.0;
   DATA[2523,19] := 2.0;
   DATA[2523,20] := 148.808;
   DATA[2523,21] := 155.4473;
   DATA[2523,22] := 1.716208;
   DATA[2523,23] := 870.7383;
   DATA[2523,24] := 2.0;
   DATA[2523,25] := 2.0;
   DATA[2523,26] := 7.874135;
   DATA[2523,27] := 144.527;
   DATA[2523,28] := 261.5355;
   DATA[2523,29] := 12.03538;
   DATA[2523,30] := 1.725711;
   DATA[2523,31] := 1.302037;
   DATA[2523,32] := 0.7352687;
   DATA[2523,33] := 0.3084905;
   DATA[2523,34] := 2.0;
   DATA[2523,35] := 250.032;
   DATA[2523,36] := 1.730048;
   DATA[2523,37] := 188.8618;
   DATA[2523,38] := 0.000128152;
   DATA[2523,39] := 1.0;
   DATA[2523,40] := 1.0;
   DATA[2524,0] := 2.433783;
   DATA[2524,1] := 868.0355;
   DATA[2524,2] := 2.0;
   DATA[2524,3] := 2.0;
   DATA[2524,4] := 262.3366;
   DATA[2524,5] := 8.39868;
   DATA[2524,6] := 329.5822;
   DATA[2524,7] := 2.452696;
   DATA[2524,8] := 2.0;
   DATA[2524,9] := 2.0;
   DATA[2524,10] := 2.0;
   DATA[2524,11] := 19.70997;
   DATA[2524,12] := 2.208116;
   DATA[2524,13] := 826.3506;
   DATA[2524,14] := 1.0;
   DATA[2524,15] := 2.0;
   DATA[2524,16] := 1.0;
   DATA[2524,17] := 1.0;
   DATA[2524,18] := 1.0;
   DATA[2524,19] := 2.0;
   DATA[2524,20] := 148.808;
   DATA[2524,21] := 155.4473;
   DATA[2524,22] := 1.716208;
   DATA[2524,23] := 870.8536;
   DATA[2524,24] := 2.0;
   DATA[2524,25] := 2.0;
   DATA[2524,26] := 7.874135;
   DATA[2524,27] := 144.527;
   DATA[2524,28] := 261.5355;
   DATA[2524,29] := 12.03538;
   DATA[2524,30] := 1.725711;
   DATA[2524,31] := 1.289356;
   DATA[2524,32] := 0.7352687;
   DATA[2524,33] := 0.3084905;
   DATA[2524,34] := 2.0;
   DATA[2524,35] := 250.032;
   DATA[2524,36] := 1.730048;
   DATA[2524,37] := 188.8618;
   DATA[2524,38] := 0.000128152;
   DATA[2524,39] := 1.0;
   DATA[2524,40] := 1.0;
   DATA[2525,0] := 2.428018;
   DATA[2525,1] := 868.271;
   DATA[2525,2] := 2.0;
   DATA[2525,3] := 2.0;
   DATA[2525,4] := 262.3366;
   DATA[2525,5] := 8.398359;
   DATA[2525,6] := 329.5822;
   DATA[2525,7] := 2.453593;
   DATA[2525,8] := 2.0;
   DATA[2525,9] := 2.0;
   DATA[2525,10] := 2.0;
   DATA[2525,11] := 19.71957;
   DATA[2525,12] := 2.208116;
   DATA[2525,13] := 826.4307;
   DATA[2525,14] := 1.0;
   DATA[2525,15] := 2.0;
   DATA[2525,16] := 1.0;
   DATA[2525,17] := 1.0;
   DATA[2525,18] := 1.0;
   DATA[2525,19] := 2.0;
   DATA[2525,20] := 148.808;
   DATA[2525,21] := 155.4473;
   DATA[2525,22] := 1.714926;
   DATA[2525,23] := 871.0844;
   DATA[2525,24] := 2.0;
   DATA[2525,25] := 2.0;
   DATA[2525,26] := 7.874135;
   DATA[2525,27] := 144.527;
   DATA[2525,28] := 261.5355;
   DATA[2525,29] := 12.03538;
   DATA[2525,30] := 1.725711;
   DATA[2525,31] := 1.289356;
   DATA[2525,32] := 0.7352687;
   DATA[2525,33] := 0.3084905;
   DATA[2525,34] := 2.0;
   DATA[2525,35] := 250.032;
   DATA[2525,36] := 1.730048;
   DATA[2525,37] := 188.8618;
   DATA[2525,38] := 0.000128152;
   DATA[2525,39] := 1.0;
   DATA[2525,40] := 1.0;
   DATA[2526,0] := 2.427377;
   DATA[2526,1] := 868.5458;
   DATA[2526,2] := 2.0;
   DATA[2526,3] := 2.0;
   DATA[2526,4] := 262.3366;
   DATA[2526,5] := 8.398359;
   DATA[2526,6] := 329.3002;
   DATA[2526,7] := 2.453593;
   DATA[2526,8] := 2.0;
   DATA[2526,9] := 2.0;
   DATA[2526,10] := 2.0;
   DATA[2526,11] := 19.72598;
   DATA[2526,12] := 2.208116;
   DATA[2526,13] := 826.4307;
   DATA[2526,14] := 1.0;
   DATA[2526,15] := 2.0;
   DATA[2526,16] := 1.0;
   DATA[2526,17] := 1.0;
   DATA[2526,18] := 1.0;
   DATA[2526,19] := 2.0;
   DATA[2526,20] := 148.808;
   DATA[2526,21] := 155.4473;
   DATA[2526,22] := 1.714926;
   DATA[2526,23] := 871.0459;
   DATA[2526,24] := 2.0;
   DATA[2526,25] := 2.0;
   DATA[2526,26] := 7.874135;
   DATA[2526,27] := 144.4758;
   DATA[2526,28] := 261.5355;
   DATA[2526,29] := 12.03538;
   DATA[2526,30] := 1.725711;
   DATA[2526,31] := 1.28167;
   DATA[2526,32] := 0.7352687;
   DATA[2526,33] := 0.3084905;
   DATA[2526,34] := 2.0;
   DATA[2526,35] := 250.032;
   DATA[2526,36] := 1.730048;
   DATA[2526,37] := 188.8618;
   DATA[2526,38] := 0.000128152;
   DATA[2526,39] := 1.0;
   DATA[2526,40] := 1.0;
   DATA[2527,0] := 2.427377;
   DATA[2527,1] := 868.7028;
   DATA[2527,2] := 2.0;
   DATA[2527,3] := 2.0;
   DATA[2527,4] := 262.3366;
   DATA[2527,5] := 8.398359;
   DATA[2527,6] := 329.3002;
   DATA[2527,7] := 2.453593;
   DATA[2527,8] := 2.0;
   DATA[2527,9] := 2.0;
   DATA[2527,10] := 2.0;
   DATA[2527,11] := 19.72598;
   DATA[2527,12] := 2.208116;
   DATA[2527,13] := 826.2305;
   DATA[2527,14] := 1.0;
   DATA[2527,15] := 2.0;
   DATA[2527,16] := 1.0;
   DATA[2527,17] := 1.0;
   DATA[2527,18] := 1.0;
   DATA[2527,19] := 2.0;
   DATA[2527,20] := 148.808;
   DATA[2527,21] := 155.4473;
   DATA[2527,22] := 1.714926;
   DATA[2527,23] := 870.8921;
   DATA[2527,24] := 2.0;
   DATA[2527,25] := 2.0;
   DATA[2527,26] := 7.874135;
   DATA[2527,27] := 144.4758;
   DATA[2527,28] := 261.5355;
   DATA[2527,29] := 12.03538;
   DATA[2527,30] := 1.725711;
   DATA[2527,31] := 1.28167;
   DATA[2527,32] := 0.7352687;
   DATA[2527,33] := 0.3084905;
   DATA[2527,34] := 2.0;
   DATA[2527,35] := 250.032;
   DATA[2527,36] := 1.730048;
   DATA[2527,37] := 188.8618;
   DATA[2527,38] := 0.000128152;
   DATA[2527,39] := 1.0;
   DATA[2527,40] := 1.0;
   DATA[2528,0] := 2.479903;
   DATA[2528,1] := 868.8206;
   DATA[2528,2] := 2.0;
   DATA[2528,3] := 2.0;
   DATA[2528,4] := 262.3366;
   DATA[2528,5] := 8.398359;
   DATA[2528,6] := 329.3002;
   DATA[2528,7] := 2.453593;
   DATA[2528,8] := 2.0;
   DATA[2528,9] := 2.0;
   DATA[2528,10] := 2.0;
   DATA[2528,11] := 19.72598;
   DATA[2528,12] := 2.208116;
   DATA[2528,13] := 826.1504;
   DATA[2528,14] := 1.0;
   DATA[2528,15] := 2.0;
   DATA[2528,16] := 1.0;
   DATA[2528,17] := 1.0;
   DATA[2528,18] := 1.0;
   DATA[2528,19] := 2.0;
   DATA[2528,20] := 148.808;
   DATA[2528,21] := 155.4473;
   DATA[2528,22] := 1.714926;
   DATA[2528,23] := 870.9305;
   DATA[2528,24] := 2.0;
   DATA[2528,25] := 2.0;
   DATA[2528,26] := 7.874135;
   DATA[2528,27] := 144.3732;
   DATA[2528,28] := 261.5355;
   DATA[2528,29] := 12.03538;
   DATA[2528,30] := 1.725711;
   DATA[2528,31] := 1.295376;
   DATA[2528,32] := 0.7352687;
   DATA[2528,33] := 0.3084905;
   DATA[2528,34] := 2.0;
   DATA[2528,35] := 250.032;
   DATA[2528,36] := 1.730048;
   DATA[2528,37] := 188.8618;
   DATA[2528,38] := 0.000128152;
   DATA[2528,39] := 1.0;
   DATA[2528,40] := 1.0;
   DATA[2529,0] := 2.528264;
   DATA[2529,1] := 868.8206;
   DATA[2529,2] := 2.0;
   DATA[2529,3] := 2.0;
   DATA[2529,4] := 262.3366;
   DATA[2529,5] := 8.398359;
   DATA[2529,6] := 329.3002;
   DATA[2529,7] := 2.453593;
   DATA[2529,8] := 2.0;
   DATA[2529,9] := 2.0;
   DATA[2529,10] := 2.0;
   DATA[2529,11] := 19.72598;
   DATA[2529,12] := 2.208116;
   DATA[2529,13] := 825.6296;
   DATA[2529,14] := 1.0;
   DATA[2529,15] := 2.0;
   DATA[2529,16] := 1.0;
   DATA[2529,17] := 1.0;
   DATA[2529,18] := 1.0;
   DATA[2529,19] := 2.0;
   DATA[2529,20] := 148.808;
   DATA[2529,21] := 155.4473;
   DATA[2529,22] := 1.714926;
   DATA[2529,23] := 870.8921;
   DATA[2529,24] := 2.0;
   DATA[2529,25] := 2.0;
   DATA[2529,26] := 7.874135;
   DATA[2529,27] := 144.3732;
   DATA[2529,28] := 261.2791;
   DATA[2529,29] := 12.03538;
   DATA[2529,30] := 1.725711;
   DATA[2529,31] := 1.301012;
   DATA[2529,32] := 0.7352687;
   DATA[2529,33] := 0.3084905;
   DATA[2529,34] := 2.0;
   DATA[2529,35] := 250.032;
   DATA[2529,36] := 1.730048;
   DATA[2529,37] := 188.8618;
   DATA[2529,38] := 0.000128152;
   DATA[2529,39] := 1.0;
   DATA[2529,40] := 1.0;
   DATA[2530,0] := 2.564776;
   DATA[2530,1] := 868.899;
   DATA[2530,2] := 2.0;
   DATA[2530,3] := 2.0;
   DATA[2530,4] := 262.3366;
   DATA[2530,5] := 8.398359;
   DATA[2530,6] := 329.4027;
   DATA[2530,7] := 2.453593;
   DATA[2530,8] := 2.0;
   DATA[2530,9] := 2.0;
   DATA[2530,10] := 2.0;
   DATA[2530,11] := 19.72598;
   DATA[2530,12] := 2.208116;
   DATA[2530,13] := 825.83;
   DATA[2530,14] := 1.0;
   DATA[2530,15] := 2.0;
   DATA[2530,16] := 1.0;
   DATA[2530,17] := 1.0;
   DATA[2530,18] := 1.0;
   DATA[2530,19] := 2.0;
   DATA[2530,20] := 148.808;
   DATA[2530,21] := 155.4473;
   DATA[2530,22] := 1.716464;
   DATA[2530,23] := 871.3535;
   DATA[2530,24] := 2.0;
   DATA[2530,25] := 2.0;
   DATA[2530,26] := 7.874135;
   DATA[2530,27] := 144.3732;
   DATA[2530,28] := 261.2791;
   DATA[2530,29] := 12.03538;
   DATA[2530,30] := 1.725711;
   DATA[2530,31] := 1.301012;
   DATA[2530,32] := 0.7352687;
   DATA[2530,33] := 0.3084905;
   DATA[2530,34] := 2.0;
   DATA[2530,35] := 250.032;
   DATA[2530,36] := 1.730048;
   DATA[2530,37] := 188.8618;
   DATA[2530,38] := 0.000128152;
   DATA[2530,39] := 1.0;
   DATA[2530,40] := 1.0;
   DATA[2531,0] := 2.600967;
   DATA[2531,1] := 868.6243;
   DATA[2531,2] := 2.0;
   DATA[2531,3] := 2.0;
   DATA[2531,4] := 262.3366;
   DATA[2531,5] := 8.398359;
   DATA[2531,6] := 329.5309;
   DATA[2531,7] := 2.45308;
   DATA[2531,8] := 2.0;
   DATA[2531,9] := 2.0;
   DATA[2531,10] := 2.0;
   DATA[2531,11] := 19.72598;
   DATA[2531,12] := 2.208116;
   DATA[2531,13] := 825.7498;
   DATA[2531,14] := 1.0;
   DATA[2531,15] := 2.0;
   DATA[2531,16] := 1.0;
   DATA[2531,17] := 1.0;
   DATA[2531,18] := 1.0;
   DATA[2531,19] := 2.0;
   DATA[2531,20] := 148.808;
   DATA[2531,21] := 155.4473;
   DATA[2531,22] := 1.717361;
   DATA[2531,23] := 871.4304;
   DATA[2531,24] := 2.0;
   DATA[2531,25] := 2.0;
   DATA[2531,26] := 7.874135;
   DATA[2531,27] := 144.3732;
   DATA[2531,28] := 261.2791;
   DATA[2531,29] := 12.03538;
   DATA[2531,30] := 1.725711;
   DATA[2531,31] := 1.292558;
   DATA[2531,32] := 0.7352687;
   DATA[2531,33] := 0.3084905;
   DATA[2531,34] := 2.0;
   DATA[2531,35] := 250.032;
   DATA[2531,36] := 1.730048;
   DATA[2531,37] := 188.8618;
   DATA[2531,38] := 0.000128152;
   DATA[2531,39] := 1.0;
   DATA[2531,40] := 1.0;
   DATA[2532,0] := 2.62723;
   DATA[2532,1] := 868.9383;
   DATA[2532,2] := 2.0;
   DATA[2532,3] := 2.0;
   DATA[2532,4] := 262.3366;
   DATA[2532,5] := 8.398359;
   DATA[2532,6] := 329.5309;
   DATA[2532,7] := 2.451415;
   DATA[2532,8] := 2.0;
   DATA[2532,9] := 2.0;
   DATA[2532,10] := 2.0;
   DATA[2532,11] := 19.70997;
   DATA[2532,12] := 2.208116;
   DATA[2532,13] := 825.4694;
   DATA[2532,14] := 1.0;
   DATA[2532,15] := 2.0;
   DATA[2532,16] := 1.0;
   DATA[2532,17] := 1.0;
   DATA[2532,18] := 1.0;
   DATA[2532,19] := 2.0;
   DATA[2532,20] := 148.808;
   DATA[2532,21] := 155.4473;
   DATA[2532,22] := 1.717361;
   DATA[2532,23] := 871.1613;
   DATA[2532,24] := 2.0;
   DATA[2532,25] := 2.0;
   DATA[2532,26] := 7.874135;
   DATA[2532,27] := 144.3732;
   DATA[2532,28] := 261.2791;
   DATA[2532,29] := 12.03538;
   DATA[2532,30] := 1.725968;
   DATA[2532,31] := 1.284488;
   DATA[2532,32] := 0.7352687;
   DATA[2532,33] := 0.3084905;
   DATA[2532,34] := 2.0;
   DATA[2532,35] := 250.032;
   DATA[2532,36] := 1.730048;
   DATA[2532,37] := 188.8618;
   DATA[2532,38] := 0.000128152;
   DATA[2532,39] := 1.0;
   DATA[2532,40] := 1.0;
   DATA[2533,0] := 2.647727;
   DATA[2533,1] := 868.7028;
   DATA[2533,2] := 2.0;
   DATA[2533,3] := 2.0;
   DATA[2533,4] := 262.3366;
   DATA[2533,5] := 8.398359;
   DATA[2533,6] := 329.5309;
   DATA[2533,7] := 2.451415;
   DATA[2533,8] := 2.0;
   DATA[2533,9] := 2.0;
   DATA[2533,10] := 2.0;
   DATA[2533,11] := 19.70037;
   DATA[2533,12] := 2.208116;
   DATA[2533,13] := 824.9487;
   DATA[2533,14] := 1.0;
   DATA[2533,15] := 2.0;
   DATA[2533,16] := 1.0;
   DATA[2533,17] := 1.0;
   DATA[2533,18] := 1.0;
   DATA[2533,19] := 2.0;
   DATA[2533,20] := 148.808;
   DATA[2533,21] := 155.4473;
   DATA[2533,22] := 1.717361;
   DATA[2533,23] := 871.1228;
   DATA[2533,24] := 2.0;
   DATA[2533,25] := 2.0;
   DATA[2533,26] := 7.874135;
   DATA[2533,27] := 144.3732;
   DATA[2533,28] := 261.2791;
   DATA[2533,29] := 12.03538;
   DATA[2533,30] := 1.726993;
   DATA[2533,31] := 1.273985;
   DATA[2533,32] := 0.7352687;
   DATA[2533,33] := 0.3084905;
   DATA[2533,34] := 2.0;
   DATA[2533,35] := 250.032;
   DATA[2533,36] := 1.730048;
   DATA[2533,37] := 188.8618;
   DATA[2533,38] := 0.000128152;
   DATA[2533,39] := 1.0;
   DATA[2533,40] := 1.0;
   DATA[2534,0] := 2.656375;
   DATA[2534,1] := 869.0168;
   DATA[2534,2] := 2.0;
   DATA[2534,3] := 2.0;
   DATA[2534,4] := 262.3366;
   DATA[2534,5] := 8.398359;
   DATA[2534,6] := 329.5309;
   DATA[2534,7] := 2.454875;
   DATA[2534,8] := 2.0;
   DATA[2534,9] := 2.0;
   DATA[2534,10] := 2.0;
   DATA[2534,11] := 19.70037;
   DATA[2534,12] := 2.208116;
   DATA[2534,13] := 824.9888;
   DATA[2534,14] := 1.0;
   DATA[2534,15] := 2.0;
   DATA[2534,16] := 1.0;
   DATA[2534,17] := 1.0;
   DATA[2534,18] := 1.0;
   DATA[2534,19] := 2.0;
   DATA[2534,20] := 148.808;
   DATA[2534,21] := 155.4473;
   DATA[2534,22] := 1.717361;
   DATA[2534,23] := 871.1228;
   DATA[2534,24] := 2.0;
   DATA[2534,25] := 2.0;
   DATA[2534,26] := 7.874135;
   DATA[2534,27] := 144.3732;
   DATA[2534,28] := 261.5355;
   DATA[2534,29] := 12.03538;
   DATA[2534,30] := 1.726993;
   DATA[2534,31] := 1.280646;
   DATA[2534,32] := 0.7352687;
   DATA[2534,33] := 0.3081062;
   DATA[2534,34] := 2.0;
   DATA[2534,35] := 250.032;
   DATA[2534,36] := 1.730048;
   DATA[2534,37] := 188.8618;
   DATA[2534,38] := 0.000128152;
   DATA[2534,39] := 1.0;
   DATA[2534,40] := 1.0;
   DATA[2535,0] := 2.656375;
   DATA[2535,1] := 868.9383;
   DATA[2535,2] := 2.0;
   DATA[2535,3] := 2.0;
   DATA[2535,4] := 262.3366;
   DATA[2535,5] := 8.398359;
   DATA[2535,6] := 329.5309;
   DATA[2535,7] := 2.454875;
   DATA[2535,8] := 2.0;
   DATA[2535,9] := 2.0;
   DATA[2535,10] := 2.0;
   DATA[2535,11] := 19.70037;
   DATA[2535,12] := 2.208116;
   DATA[2535,13] := 824.6684;
   DATA[2535,14] := 1.0;
   DATA[2535,15] := 2.0;
   DATA[2535,16] := 1.0;
   DATA[2535,17] := 1.0;
   DATA[2535,18] := 1.0;
   DATA[2535,19] := 2.0;
   DATA[2535,20] := 148.808;
   DATA[2535,21] := 155.4473;
   DATA[2535,22] := 1.717361;
   DATA[2535,23] := 871.0844;
   DATA[2535,24] := 2.0;
   DATA[2535,25] := 2.0;
   DATA[2535,26] := 7.874135;
   DATA[2535,27] := 144.3732;
   DATA[2535,28] := 261.5996;
   DATA[2535,29] := 12.03538;
   DATA[2535,30] := 1.726993;
   DATA[2535,31] := 1.286666;
   DATA[2535,32] := 0.7352687;
   DATA[2535,33] := 0.3081062;
   DATA[2535,34] := 2.0;
   DATA[2535,35] := 250.032;
   DATA[2535,36] := 1.730048;
   DATA[2535,37] := 188.958;
   DATA[2535,38] := 0.000128152;
   DATA[2535,39] := 1.0;
   DATA[2535,40] := 1.0;
   DATA[2536,0] := 2.628511;
   DATA[2536,1] := 869.4094;
   DATA[2536,2] := 2.0;
   DATA[2536,3] := 2.0;
   DATA[2536,4] := 262.3366;
   DATA[2536,5] := 8.398359;
   DATA[2536,6] := 329.5309;
   DATA[2536,7] := 2.454875;
   DATA[2536,8] := 2.0;
   DATA[2536,9] := 2.0;
   DATA[2536,10] := 2.0;
   DATA[2536,11] := 19.70037;
   DATA[2536,12] := 2.206835;
   DATA[2536,13] := 824.6684;
   DATA[2536,14] := 1.0;
   DATA[2536,15] := 2.0;
   DATA[2536,16] := 1.0;
   DATA[2536,17] := 1.0;
   DATA[2536,18] := 1.0;
   DATA[2536,19] := 2.0;
   DATA[2536,20] := 148.808;
   DATA[2536,21] := 155.4473;
   DATA[2536,22] := 1.717361;
   DATA[2536,23] := 871.2766;
   DATA[2536,24] := 2.0;
   DATA[2536,25] := 2.0;
   DATA[2536,26] := 7.872533;
   DATA[2536,27] := 144.3732;
   DATA[2536,28] := 261.5996;
   DATA[2536,29] := 12.03538;
   DATA[2536,30] := 1.726993;
   DATA[2536,31] := 1.291789;
   DATA[2536,32] := 0.7352687;
   DATA[2536,33] := 0.3081062;
   DATA[2536,34] := 2.0;
   DATA[2536,35] := 250.0961;
   DATA[2536,36] := 1.730048;
   DATA[2536,37] := 189.1182;
   DATA[2536,38] := 0.000128152;
   DATA[2536,39] := 1.0;
   DATA[2536,40] := 1.0;
   DATA[2537,0] := 2.614419;
   DATA[2537,1] := 869.6448;
   DATA[2537,2] := 2.0;
   DATA[2537,3] := 2.0;
   DATA[2537,4] := 262.3366;
   DATA[2537,5] := 8.398359;
   DATA[2537,6] := 329.2745;
   DATA[2537,7] := 2.452952;
   DATA[2537,8] := 2.0;
   DATA[2537,9] := 2.0;
   DATA[2537,10] := 2.0;
   DATA[2537,11] := 19.70037;
   DATA[2537,12] := 2.20645;
   DATA[2537,13] := 824.6684;
   DATA[2537,14] := 1.0;
   DATA[2537,15] := 2.0;
   DATA[2537,16] := 1.0;
   DATA[2537,17] := 1.0;
   DATA[2537,18] := 1.0;
   DATA[2537,19] := 2.0;
   DATA[2537,20] := 148.808;
   DATA[2537,21] := 155.4473;
   DATA[2537,22] := 1.71813;
   DATA[2537,23] := 871.3535;
   DATA[2537,24] := 2.0;
   DATA[2537,25] := 2.0;
   DATA[2537,26] := 7.872533;
   DATA[2537,27] := 144.3732;
   DATA[2537,28] := 261.5355;
   DATA[2537,29] := 12.03538;
   DATA[2537,30] := 1.727378;
   DATA[2537,31] := 1.291789;
   DATA[2537,32] := 0.7352687;
   DATA[2537,33] := 0.3081062;
   DATA[2537,34] := 2.0;
   DATA[2537,35] := 250.2403;
   DATA[2537,36] := 1.730048;
   DATA[2537,37] := 189.1182;
   DATA[2537,38] := 0.000128152;
   DATA[2537,39] := 1.0;
   DATA[2537,40] := 1.0;
   DATA[2538,0] := 2.609935;
   DATA[2538,1] := 869.0561;
   DATA[2538,2] := 2.0;
   DATA[2538,3] := 2.0;
   DATA[2538,4] := 262.3366;
   DATA[2538,5] := 8.398359;
   DATA[2538,6] := 329.2745;
   DATA[2538,7] := 2.452952;
   DATA[2538,8] := 2.0;
   DATA[2538,9] := 2.0;
   DATA[2538,10] := 2.0;
   DATA[2538,11] := 19.70037;
   DATA[2538,12] := 2.20645;
   DATA[2538,13] := 824.428;
   DATA[2538,14] := 1.0;
   DATA[2538,15] := 2.0;
   DATA[2538,16] := 1.0;
   DATA[2538,17] := 1.0;
   DATA[2538,18] := 1.0;
   DATA[2538,19] := 2.0;
   DATA[2538,20] := 148.808;
   DATA[2538,21] := 155.4473;
   DATA[2538,22] := 1.718515;
   DATA[2538,23] := 871.2382;
   DATA[2538,24] := 2.0;
   DATA[2538,25] := 2.0;
   DATA[2538,26] := 7.872533;
   DATA[2538,27] := 144.3732;
   DATA[2538,28] := 261.4073;
   DATA[2538,29] := 12.03538;
   DATA[2538,30] := 1.728275;
   DATA[2538,31] := 1.285001;
   DATA[2538,32] := 0.7352687;
   DATA[2538,33] := 0.3081062;
   DATA[2538,34] := 2.0;
   DATA[2538,35] := 250.3365;
   DATA[2538,36] := 1.681991;
   DATA[2538,37] := 189.1182;
   DATA[2538,38] := 0.000128152;
   DATA[2538,39] := 1.0;
   DATA[2538,40] := 1.0;
   DATA[2539,0] := 2.595522;
   DATA[2539,1] := 869.2131;
   DATA[2539,2] := 2.0;
   DATA[2539,3] := 2.0;
   DATA[2539,4] := 262.3366;
   DATA[2539,5] := 8.398359;
   DATA[2539,6] := 329.2745;
   DATA[2539,7] := 2.455515;
   DATA[2539,8] := 2.0;
   DATA[2539,9] := 2.0;
   DATA[2539,10] := 2.0;
   DATA[2539,11] := 19.70037;
   DATA[2539,12] := 2.20645;
   DATA[2539,13] := 824.6283;
   DATA[2539,14] := 1.0;
   DATA[2539,15] := 2.0;
   DATA[2539,16] := 1.0;
   DATA[2539,17] := 1.0;
   DATA[2539,18] := 1.0;
   DATA[2539,19] := 2.0;
   DATA[2539,20] := 148.808;
   DATA[2539,21] := 155.4473;
   DATA[2539,22] := 1.721975;
   DATA[2539,23] := 870.969;
   DATA[2539,24] := 2.0;
   DATA[2539,25] := 2.0;
   DATA[2539,26] := 7.872533;
   DATA[2539,27] := 144.3732;
   DATA[2539,28] := 261.4073;
   DATA[2539,29] := 12.03538;
   DATA[2539,30] := 1.7293;
   DATA[2539,31] := 1.286666;
   DATA[2539,32] := 0.7352687;
   DATA[2539,33] := 0.3081062;
   DATA[2539,34] := 2.0;
   DATA[2539,35] := 250.3365;
   DATA[2539,36] := 1.601897;
   DATA[2539,37] := 189.1182;
   DATA[2539,38] := 0.000128152;
   DATA[2539,39] := 1.0;
   DATA[2539,40] := 1.0;
   DATA[2540,0] := 2.587195;
   DATA[2540,1] := 868.6635;
   DATA[2540,2] := 2.0;
   DATA[2540,3] := 2.0;
   DATA[2540,4] := 262.3366;
   DATA[2540,5] := 8.395475;
   DATA[2540,6] := 329.2745;
   DATA[2540,7] := 2.455515;
   DATA[2540,8] := 2.0;
   DATA[2540,9] := 2.0;
   DATA[2540,10] := 2.0;
   DATA[2540,11] := 19.70037;
   DATA[2540,12] := 2.20645;
   DATA[2540,13] := 824.8286;
   DATA[2540,14] := 1.0;
   DATA[2540,15] := 2.0;
   DATA[2540,16] := 1.0;
   DATA[2540,17] := 1.0;
   DATA[2540,18] := 1.0;
   DATA[2540,19] := 2.0;
   DATA[2540,20] := 148.808;
   DATA[2540,21] := 155.4473;
   DATA[2540,22] := 1.721975;
   DATA[2540,23] := 871.0844;
   DATA[2540,24] := 2.0;
   DATA[2540,25] := 2.0;
   DATA[2540,26] := 7.872533;
   DATA[2540,27] := 144.3732;
   DATA[2540,28] := 261.4073;
   DATA[2540,29] := 12.03538;
   DATA[2540,30] := 1.7293;
   DATA[2540,31] := 1.279749;
   DATA[2540,32] := 0.7352687;
   DATA[2540,33] := 0.3086827;
   DATA[2540,34] := 2.0;
   DATA[2540,35] := 250.3365;
   DATA[2540,36] := 1.601897;
   DATA[2540,37] := 189.1182;
   DATA[2540,38] := 0.000128152;
   DATA[2540,39] := 1.0;
   DATA[2540,40] := 1.0;
   DATA[2541,0] := 2.561253;
   DATA[2541,1] := 868.5458;
   DATA[2541,2] := 2.0;
   DATA[2541,3] := 2.0;
   DATA[2541,4] := 262.3366;
   DATA[2541,5] := 8.395475;
   DATA[2541,6] := 329.454;
   DATA[2541,7] := 2.452568;
   DATA[2541,8] := 2.0;
   DATA[2541,9] := 2.0;
   DATA[2541,10] := 2.0;
   DATA[2541,11] := 19.74198;
   DATA[2541,12] := 2.20645;
   DATA[2541,13] := 825.1891;
   DATA[2541,14] := 1.0;
   DATA[2541,15] := 2.0;
   DATA[2541,16] := 1.0;
   DATA[2541,17] := 1.0;
   DATA[2541,18] := 1.0;
   DATA[2541,19] := 2.0;
   DATA[2541,20] := 148.808;
   DATA[2541,21] := 155.4473;
   DATA[2541,22] := 1.721975;
   DATA[2541,23] := 870.8921;
   DATA[2541,24] := 2.0;
   DATA[2541,25] := 2.0;
   DATA[2541,26] := 7.874455;
   DATA[2541,27] := 144.3732;
   DATA[2541,28] := 261.4073;
   DATA[2541,29] := 12.03538;
   DATA[2541,30] := 1.7293;
   DATA[2541,31] := 1.282567;
   DATA[2541,32] := 0.7352687;
   DATA[2541,33] := 0.3071454;
   DATA[2541,34] := 2.0;
   DATA[2541,35] := 250.3365;
   DATA[2541,36] := 1.681991;
   DATA[2541,37] := 189.1182;
   DATA[2541,38] := 0.000128152;
   DATA[2541,39] := 1.0;
   DATA[2541,40] := 1.0;
   DATA[2542,0] := 2.544278;
   DATA[2542,1] := 868.6635;
   DATA[2542,2] := 2.0;
   DATA[2542,3] := 2.0;
   DATA[2542,4] := 262.3366;
   DATA[2542,5] := 8.395475;
   DATA[2542,6] := 329.454;
   DATA[2542,7] := 2.451799;
   DATA[2542,8] := 2.0;
   DATA[2542,9] := 2.0;
   DATA[2542,10] := 2.0;
   DATA[2542,11] := 19.74198;
   DATA[2542,12] := 2.208628;
   DATA[2542,13] := 825.0689;
   DATA[2542,14] := 1.0;
   DATA[2542,15] := 2.0;
   DATA[2542,16] := 1.0;
   DATA[2542,17] := 1.0;
   DATA[2542,18] := 1.0;
   DATA[2542,19] := 2.0;
   DATA[2542,20] := 148.808;
   DATA[2542,21] := 155.4473;
   DATA[2542,22] := 1.72095;
   DATA[2542,23] := 871.2766;
   DATA[2542,24] := 2.0;
   DATA[2542,25] := 2.0;
   DATA[2542,26] := 7.874455;
   DATA[2542,27] := 144.3732;
   DATA[2542,28] := 261.4073;
   DATA[2542,29] := 12.03538;
   DATA[2542,30] := 1.7293;
   DATA[2542,31] := 1.291789;
   DATA[2542,32] := 0.7352687;
   DATA[2542,33] := 0.3064407;
   DATA[2542,34] := 2.0;
   DATA[2542,35] := 250.3365;
   DATA[2542,36] := 1.681991;
   DATA[2542,37] := 189.2143;
   DATA[2542,38] := 0.000128152;
   DATA[2542,39] := 1.0;
   DATA[2542,40] := 1.0;
   DATA[2543,0] := 2.528264;
   DATA[2543,1] := 869.0168;
   DATA[2543,2] := 2.0;
   DATA[2543,3] := 2.0;
   DATA[2543,4] := 262.3366;
   DATA[2543,5] := 8.395475;
   DATA[2543,6] := 329.454;
   DATA[2543,7] := 2.451799;
   DATA[2543,8] := 2.0;
   DATA[2543,9] := 2.0;
   DATA[2543,10] := 2.0;
   DATA[2543,11] := 19.74198;
   DATA[2543,12] := 2.210037;
   DATA[2543,13] := 825.2291;
   DATA[2543,14] := 1.0;
   DATA[2543,15] := 2.0;
   DATA[2543,16] := 1.0;
   DATA[2543,17] := 1.0;
   DATA[2543,18] := 1.0;
   DATA[2543,19] := 2.0;
   DATA[2543,20] := 148.808;
   DATA[2543,21] := 155.4473;
   DATA[2543,22] := 1.720437;
   DATA[2543,23] := 871.4304;
   DATA[2543,24] := 2.0;
   DATA[2543,25] := 2.0;
   DATA[2543,26] := 7.874455;
   DATA[2543,27] := 144.3732;
   DATA[2543,28] := 261.4073;
   DATA[2543,29] := 12.03538;
   DATA[2543,30] := 1.7293;
   DATA[2543,31] := 1.291789;
   DATA[2543,32] := 0.7352687;
   DATA[2543,33] := 0.3064407;
   DATA[2543,34] := 2.0;
   DATA[2543,35] := 250.3365;
   DATA[2543,36] := 1.681991;
   DATA[2543,37] := 189.2143;
   DATA[2543,38] := 0.000128152;
   DATA[2543,39] := 1.0;
   DATA[2543,40] := 1.0;
   DATA[2544,0] := 2.512891;
   DATA[2544,1] := 868.8598;
   DATA[2544,2] := 2.0;
   DATA[2544,3] := 2.0;
   DATA[2544,4] := 262.3366;
   DATA[2544,5] := 8.395475;
   DATA[2544,6] := 329.454;
   DATA[2544,7] := 2.451799;
   DATA[2544,8] := 2.0;
   DATA[2544,9] := 2.0;
   DATA[2544,10] := 2.0;
   DATA[2544,11] := 19.70677;
   DATA[2544,12] := 2.210166;
   DATA[2544,13] := 825.3493;
   DATA[2544,14] := 1.0;
   DATA[2544,15] := 2.0;
   DATA[2544,16] := 1.0;
   DATA[2544,17] := 1.0;
   DATA[2544,18] := 1.0;
   DATA[2544,19] := 2.0;
   DATA[2544,20] := 148.808;
   DATA[2544,21] := 155.4473;
   DATA[2544,22] := 1.71813;
   DATA[2544,23] := 871.3151;
   DATA[2544,24] := 2.0;
   DATA[2544,25] := 2.0;
   DATA[2544,26] := 7.874455;
   DATA[2544,27] := 144.3732;
   DATA[2544,28] := 261.4073;
   DATA[2544,29] := 12.03538;
   DATA[2544,30] := 1.7293;
   DATA[2544,31] := 1.291789;
   DATA[2544,32] := 0.7352687;
   DATA[2544,33] := 0.3064407;
   DATA[2544,34] := 2.0;
   DATA[2544,35] := 250.3365;
   DATA[2544,36] := 1.681991;
   DATA[2544,37] := 189.2143;
   DATA[2544,38] := 0.000128152;
   DATA[2544,39] := 1.0;
   DATA[2544,40] := 1.0;
   DATA[2545,0] := 2.501041;
   DATA[2545,1] := 869.1346;
   DATA[2545,2] := 2.0;
   DATA[2545,3] := 2.0;
   DATA[2545,4] := 262.3366;
   DATA[2545,5] := 8.395475;
   DATA[2545,6] := 329.454;
   DATA[2545,7] := 2.451799;
   DATA[2545,8] := 2.0;
   DATA[2545,9] := 2.0;
   DATA[2545,10] := 2.0;
   DATA[2545,11] := 19.70677;
   DATA[2545,12] := 2.210166;
   DATA[2545,13] := 825.7498;
   DATA[2545,14] := 1.0;
   DATA[2545,15] := 2.0;
   DATA[2545,16] := 1.0;
   DATA[2545,17] := 1.0;
   DATA[2545,18] := 1.0;
   DATA[2545,19] := 2.0;
   DATA[2545,20] := 148.808;
   DATA[2545,21] := 155.4473;
   DATA[2545,22] := 1.71813;
   DATA[2545,23] := 871.738;
   DATA[2545,24] := 2.0;
   DATA[2545,25] := 2.0;
   DATA[2545,26] := 7.874455;
   DATA[2545,27] := 144.3732;
   DATA[2545,28] := 261.4073;
   DATA[2545,29] := 12.03538;
   DATA[2545,30] := 1.7293;
   DATA[2545,31] := 1.291789;
   DATA[2545,32] := 0.7352687;
   DATA[2545,33] := 0.3064407;
   DATA[2545,34] := 2.0;
   DATA[2545,35] := 250.3365;
   DATA[2545,36] := 1.730048;
   DATA[2545,37] := 189.2143;
   DATA[2545,38] := 0.000128152;
   DATA[2545,39] := 1.0;
   DATA[2545,40] := 1.0;
   DATA[2546,0] := 2.484707;
   DATA[2546,1] := 869.0953;
   DATA[2546,2] := 2.0;
   DATA[2546,3] := 2.0;
   DATA[2546,4] := 262.3366;
   DATA[2546,5] := 8.395475;
   DATA[2546,6] := 329.454;
   DATA[2546,7] := 2.451799;
   DATA[2546,8] := 2.0;
   DATA[2546,9] := 2.0;
   DATA[2546,10] := 2.0;
   DATA[2546,11] := 19.67476;
   DATA[2546,12] := 2.210166;
   DATA[2546,13] := 825.6296;
   DATA[2546,14] := 1.0;
   DATA[2546,15] := 2.0;
   DATA[2546,16] := 1.0;
   DATA[2546,17] := 1.0;
   DATA[2546,18] := 1.0;
   DATA[2546,19] := 2.0;
   DATA[2546,20] := 148.808;
   DATA[2546,21] := 155.4473;
   DATA[2546,22] := 1.71813;
   DATA[2546,23] := 871.9303;
   DATA[2546,24] := 2.0;
   DATA[2546,25] := 2.0;
   DATA[2546,26] := 7.874455;
   DATA[2546,27] := 144.3732;
   DATA[2546,28] := 261.5996;
   DATA[2546,29] := 12.03538;
   DATA[2546,30] := 1.7293;
   DATA[2546,31] := 1.291789;
   DATA[2546,32] := 0.7352687;
   DATA[2546,33] := 0.3064407;
   DATA[2546,34] := 2.0;
   DATA[2546,35] := 250.3365;
   DATA[2546,36] := 1.730048;
   DATA[2546,37] := 189.2143;
   DATA[2546,38] := 0.000128152;
   DATA[2546,39] := 1.0;
   DATA[2546,40] := 1.0;
   DATA[2547,0] := 2.471255;
   DATA[2547,1] := 869.2916;
   DATA[2547,2] := 2.0;
   DATA[2547,3] := 2.0;
   DATA[2547,4] := 262.3366;
   DATA[2547,5] := 8.395475;
   DATA[2547,6] := 329.454;
   DATA[2547,7] := 2.449877;
   DATA[2547,8] := 2.0;
   DATA[2547,9] := 2.0;
   DATA[2547,10] := 2.0;
   DATA[2547,11] := 19.62033;
   DATA[2547,12] := 2.212728;
   DATA[2547,13] := 826.0703;
   DATA[2547,14] := 1.0;
   DATA[2547,15] := 2.0;
   DATA[2547,16] := 1.0;
   DATA[2547,17] := 1.0;
   DATA[2547,18] := 1.0;
   DATA[2547,19] := 2.0;
   DATA[2547,20] := 148.808;
   DATA[2547,21] := 155.4473;
   DATA[2547,22] := 1.71813;
   DATA[2547,23] := 872.0841;
   DATA[2547,24] := 2.0;
   DATA[2547,25] := 2.0;
   DATA[2547,26] := 7.874455;
   DATA[2547,27] := 144.3732;
   DATA[2547,28] := 261.5996;
   DATA[2547,29] := 12.03538;
   DATA[2547,30] := 1.7293;
   DATA[2547,31] := 1.302293;
   DATA[2547,32] := 0.7352687;
   DATA[2547,33] := 0.3064407;
   DATA[2547,34] := 2.0;
   DATA[2547,35] := 250.3365;
   DATA[2547,36] := 1.730048;
   DATA[2547,37] := 189.1983;
   DATA[2547,38] := 0.000128152;
   DATA[2547,39] := 1.0;
   DATA[2547,40] := 1.0;
   DATA[2548,0] := 2.454601;
   DATA[2548,1] := 869.6056;
   DATA[2548,2] := 2.0;
   DATA[2548,3] := 2.0;
   DATA[2548,4] := 262.3366;
   DATA[2548,5] := 8.395475;
   DATA[2548,6] := 329.454;
   DATA[2548,7] := 2.448851;
   DATA[2548,8] := 2.0;
   DATA[2548,9] := 2.0;
   DATA[2548,10] := 2.0;
   DATA[2548,11] := 19.60433;
   DATA[2548,12] := 2.213368;
   DATA[2548,13] := 825.9501;
   DATA[2548,14] := 1.0;
   DATA[2548,15] := 2.0;
   DATA[2548,16] := 1.0;
   DATA[2548,17] := 1.0;
   DATA[2548,18] := 1.0;
   DATA[2548,19] := 2.0;
   DATA[2548,20] := 148.808;
   DATA[2548,21] := 155.4473;
   DATA[2548,22] := 1.71813;
   DATA[2548,23] := 872.1995;
   DATA[2548,24] := 2.0;
   DATA[2548,25] := 2.0;
   DATA[2548,26] := 7.874455;
   DATA[2548,27] := 144.3732;
   DATA[2548,28] := 261.5996;
   DATA[2548,29] := 12.03538;
   DATA[2548,30] := 1.7293;
   DATA[2548,31] := 1.312028;
   DATA[2548,32] := 0.7352687;
   DATA[2548,33] := 0.3065048;
   DATA[2548,34] := 2.0;
   DATA[2548,35] := 250.3365;
   DATA[2548,36] := 1.730048;
   DATA[2548,37] := 189.1182;
   DATA[2548,38] := 0.000128152;
   DATA[2548,39] := 1.0;
   DATA[2548,40] := 1.0;
   DATA[2549,0] := 2.439548;
   DATA[2549,1] := 869.1346;
   DATA[2549,2] := 2.0;
   DATA[2549,3] := 2.0;
   DATA[2549,4] := 262.3366;
   DATA[2549,5] := 8.395475;
   DATA[2549,6] := 329.454;
   DATA[2549,7] := 2.448851;
   DATA[2549,8] := 2.0;
   DATA[2549,9] := 2.0;
   DATA[2549,10] := 2.0;
   DATA[2549,11] := 19.66835;
   DATA[2549,12] := 2.213368;
   DATA[2549,13] := 826.2305;
   DATA[2549,14] := 1.0;
   DATA[2549,15] := 2.0;
   DATA[2549,16] := 1.0;
   DATA[2549,17] := 1.0;
   DATA[2549,18] := 1.0;
   DATA[2549,19] := 2.0;
   DATA[2549,20] := 148.808;
   DATA[2549,21] := 155.3961;
   DATA[2549,22] := 1.71813;
   DATA[2549,23] := 872.3917;
   DATA[2549,24] := 2.0;
   DATA[2549,25] := 2.0;
   DATA[2549,26] := 7.874455;
   DATA[2549,27] := 144.3989;
   DATA[2549,28] := 261.5996;
   DATA[2549,29] := 12.03538;
   DATA[2549,30] := 1.7293;
   DATA[2549,31] := 1.312668;
   DATA[2549,32] := 0.7352687;
   DATA[2549,33] := 0.3068251;
   DATA[2549,34] := 2.0;
   DATA[2549,35] := 250.1122;
   DATA[2549,36] := 1.649953;
   DATA[2549,37] := 188.9419;
   DATA[2549,38] := 0.000128152;
   DATA[2549,39] := 1.0;
   DATA[2549,40] := 1.0;
   DATA[2550,0] := 2.438267;
   DATA[2550,1] := 869.0168;
   DATA[2550,2] := 2.0;
   DATA[2550,3] := 2.0;
   DATA[2550,4] := 262.3366;
   DATA[2550,5] := 8.395475;
   DATA[2550,6] := 329.454;
   DATA[2550,7] := 2.451671;
   DATA[2550,8] := 2.0;
   DATA[2550,9] := 2.0;
   DATA[2550,10] := 2.0;
   DATA[2550,11] := 19.70997;
   DATA[2550,12] := 2.211831;
   DATA[2550,13] := 826.3506;
   DATA[2550,14] := 1.0;
   DATA[2550,15] := 2.0;
   DATA[2550,16] := 1.0;
   DATA[2550,17] := 1.0;
   DATA[2550,18] := 1.0;
   DATA[2550,19] := 2.0;
   DATA[2550,20] := 148.808;
   DATA[2550,21] := 155.191;
   DATA[2550,22] := 1.71813;
   DATA[2550,23] := 872.5839;
   DATA[2550,24] := 2.0;
   DATA[2550,25] := 2.0;
   DATA[2550,26] := 7.874455;
   DATA[2550,27] := 144.4758;
   DATA[2550,28] := 261.5996;
   DATA[2550,29] := 12.03538;
   DATA[2550,30] := 1.7293;
   DATA[2550,31] := 1.306648;
   DATA[2550,32] := 0.7352687;
   DATA[2550,33] := 0.3068251;
   DATA[2550,34] := 2.0;
   DATA[2550,35] := 250.1122;
   DATA[2550,36] := 1.649953;
   DATA[2550,37] := 188.8779;
   DATA[2550,38] := 0.000128152;
   DATA[2550,39] := 1.0;
   DATA[2550,40] := 1.0;
   DATA[2551,0] := 2.438267;
   DATA[2551,1] := 869.2523;
   DATA[2551,2] := 2.0;
   DATA[2551,3] := 2.0;
   DATA[2551,4] := 262.3366;
   DATA[2551,5] := 8.395475;
   DATA[2551,6] := 329.454;
   DATA[2551,7] := 2.451671;
   DATA[2551,8] := 2.0;
   DATA[2551,9] := 2.0;
   DATA[2551,10] := 2.0;
   DATA[2551,11] := 19.70997;
   DATA[2551,12] := 2.210934;
   DATA[2551,13] := 826.4307;
   DATA[2551,14] := 1.0;
   DATA[2551,15] := 2.0;
   DATA[2551,16] := 1.0;
   DATA[2551,17] := 1.0;
   DATA[2551,18] := 1.0;
   DATA[2551,19] := 2.0;
   DATA[2551,20] := 148.808;
   DATA[2551,21] := 155.191;
   DATA[2551,22] := 1.71813;
   DATA[2551,23] := 872.8531;
   DATA[2551,24] := 2.0;
   DATA[2551,25] := 2.0;
   DATA[2551,26] := 7.874455;
   DATA[2551,27] := 144.4758;
   DATA[2551,28] := 261.5996;
   DATA[2551,29] := 12.03538;
   DATA[2551,30] := 1.728531;
   DATA[2551,31] := 1.306776;
   DATA[2551,32] := 0.7352687;
   DATA[2551,33] := 0.3068251;
   DATA[2551,34] := 2.0;
   DATA[2551,35] := 250.1122;
   DATA[2551,36] := 1.649953;
   DATA[2551,37] := 188.8779;
   DATA[2551,38] := 0.000128152;
   DATA[2551,39] := 1.0;
   DATA[2551,40] := 1.0;
   DATA[2552,0] := 2.438267;
   DATA[2552,1] := 869.2523;
   DATA[2552,2] := 2.0;
   DATA[2552,3] := 2.0;
   DATA[2552,4] := 262.3366;
   DATA[2552,5] := 8.395475;
   DATA[2552,6] := 329.454;
   DATA[2552,7] := 2.451671;
   DATA[2552,8] := 2.0;
   DATA[2552,9] := 2.0;
   DATA[2552,10] := 2.0;
   DATA[2552,11] := 19.70997;
   DATA[2552,12] := 2.210934;
   DATA[2552,13] := 826.4307;
   DATA[2552,14] := 1.0;
   DATA[2552,15] := 2.0;
   DATA[2552,16] := 1.0;
   DATA[2552,17] := 1.0;
   DATA[2552,18] := 1.0;
   DATA[2552,19] := 2.0;
   DATA[2552,20] := 148.808;
   DATA[2552,21] := 155.191;
   DATA[2552,22] := 1.71813;
   DATA[2552,23] := 872.8531;
   DATA[2552,24] := 2.0;
   DATA[2552,25] := 2.0;
   DATA[2552,26] := 7.874455;
   DATA[2552,27] := 144.4758;
   DATA[2552,28] := 261.5996;
   DATA[2552,29] := 12.03538;
   DATA[2552,30] := 1.728531;
   DATA[2552,31] := 1.306776;
   DATA[2552,32] := 0.7352687;
   DATA[2552,33] := 0.3068251;
   DATA[2552,34] := 2.0;
   DATA[2552,35] := 250.1122;
   DATA[2552,36] := 1.649953;
   DATA[2552,37] := 188.8779;
   DATA[2552,38] := 0.000128152;
   DATA[2552,39] := 1.0;
   DATA[2552,40] := 1.0;
   DATA[2553,0] := 2.479262;
   DATA[2553,1] := 869.1346;
   DATA[2553,2] := 2.0;
   DATA[2553,3] := 2.0;
   DATA[2553,4] := 262.3366;
   DATA[2553,5] := 8.393873;
   DATA[2553,6] := 329.454;
   DATA[2553,7] := 2.451671;
   DATA[2553,8] := 2.0;
   DATA[2553,9] := 2.0;
   DATA[2553,10] := 2.0;
   DATA[2553,11] := 19.70997;
   DATA[2553,12] := 2.210934;
   DATA[2553,13] := 826.7912;
   DATA[2553,14] := 1.0;
   DATA[2553,15] := 2.0;
   DATA[2553,16] := 1.0;
   DATA[2553,17] := 1.0;
   DATA[2553,18] := 1.0;
   DATA[2553,19] := 2.0;
   DATA[2553,20] := 148.808;
   DATA[2553,21] := 155.191;
   DATA[2553,22] := 1.71813;
   DATA[2553,23] := 873.5837;
   DATA[2553,24] := 2.0;
   DATA[2553,25] := 2.0;
   DATA[2553,26] := 7.874455;
   DATA[2553,27] := 144.4758;
   DATA[2553,28] := 261.5996;
   DATA[2553,29] := 12.03538;
   DATA[2553,30] := 1.726352;
   DATA[2553,31] := 1.293967;
   DATA[2553,32] := 0.7352687;
   DATA[2553,33] := 0.3071454;
   DATA[2553,34] := 2.0;
   DATA[2553,35] := 250.032;
   DATA[2553,36] := 1.649953;
   DATA[2553,37] := 188.8779;
   DATA[2553,38] := 0.000128152;
   DATA[2553,39] := 1.0;
   DATA[2553,40] := 1.0;
   DATA[2554,0] := 2.514493;
   DATA[2554,1] := 869.1346;
   DATA[2554,2] := 2.0;
   DATA[2554,3] := 2.0;
   DATA[2554,4] := 262.3366;
   DATA[2554,5] := 8.393873;
   DATA[2554,6] := 329.454;
   DATA[2554,7] := 2.451671;
   DATA[2554,8] := 2.0;
   DATA[2554,9] := 2.0;
   DATA[2554,10] := 2.0;
   DATA[2554,11] := 19.70997;
   DATA[2554,12] := 2.210294;
   DATA[2554,13] := 826.5509;
   DATA[2554,14] := 1.0;
   DATA[2554,15] := 2.0;
   DATA[2554,16] := 1.0;
   DATA[2554,17] := 1.0;
   DATA[2554,18] := 1.0;
   DATA[2554,19] := 2.0;
   DATA[2554,20] := 148.808;
   DATA[2554,21] := 155.191;
   DATA[2554,22] := 1.71813;
   DATA[2554,23] := 873.8144;
   DATA[2554,24] := 2.0;
   DATA[2554,25] := 2.0;
   DATA[2554,26] := 7.874455;
   DATA[2554,27] := 144.4758;
   DATA[2554,28] := 261.5996;
   DATA[2554,29] := 12.03538;
   DATA[2554,30] := 1.726224;
   DATA[2554,31] := 1.291533;
   DATA[2554,32] := 0.7352687;
   DATA[2554,33] := 0.3084265;
   DATA[2554,34] := 2.0;
   DATA[2554,35] := 250.032;
   DATA[2554,36] := 1.649953;
   DATA[2554,37] := 188.8779;
   DATA[2554,38] := 0.000128152;
   DATA[2554,39] := 1.0;
   DATA[2554,40] := 1.0;
   DATA[2555,0] := 2.558691;
   DATA[2555,1] := 869.2523;
   DATA[2555,2] := 2.0;
   DATA[2555,3] := 2.0;
   DATA[2555,4] := 262.3366;
   DATA[2555,5] := 8.393873;
   DATA[2555,6] := 329.454;
   DATA[2555,7] := 2.451671;
   DATA[2555,8] := 2.0;
   DATA[2555,9] := 2.0;
   DATA[2555,10] := 2.0;
   DATA[2555,11] := 19.70997;
   DATA[2555,12] := 2.209525;
   DATA[2555,13] := 826.3907;
   DATA[2555,14] := 1.0;
   DATA[2555,15] := 2.0;
   DATA[2555,16] := 1.0;
   DATA[2555,17] := 1.0;
   DATA[2555,18] := 1.0;
   DATA[2555,19] := 2.0;
   DATA[2555,20] := 148.808;
   DATA[2555,21] := 155.191;
   DATA[2555,22] := 1.71813;
   DATA[2555,23] := 873.5452;
   DATA[2555,24] := 2.0;
   DATA[2555,25] := 2.0;
   DATA[2555,26] := 7.871251;
   DATA[2555,27] := 144.4758;
   DATA[2555,28] := 261.5996;
   DATA[2555,29] := 12.03538;
   DATA[2555,30] := 1.726224;
   DATA[2555,31] := 1.283464;
   DATA[2555,32] := 0.7352687;
   DATA[2555,33] := 0.3084265;
   DATA[2555,34] := 2.0;
   DATA[2555,35] := 250.032;
   DATA[2555,36] := 1.649953;
   DATA[2555,37] := 188.8779;
   DATA[2555,38] := 0.000128152;
   DATA[2555,39] := 1.0;
   DATA[2555,40] := 1.0;
   DATA[2556,0] := 2.587516;
   DATA[2556,1] := 868.9383;
   DATA[2556,2] := 2.0;
   DATA[2556,3] := 2.0;
   DATA[2556,4] := 262.3366;
   DATA[2556,5] := 8.393873;
   DATA[2556,6] := 329.454;
   DATA[2556,7] := 2.452568;
   DATA[2556,8] := 2.0;
   DATA[2556,9] := 2.0;
   DATA[2556,10] := 2.0;
   DATA[2556,11] := 19.70997;
   DATA[2556,12] := 2.209525;
   DATA[2556,13] := 826.6711;
   DATA[2556,14] := 1.0;
   DATA[2556,15] := 2.0;
   DATA[2556,16] := 1.0;
   DATA[2556,17] := 1.0;
   DATA[2556,18] := 1.0;
   DATA[2556,19] := 2.0;
   DATA[2556,20] := 148.808;
   DATA[2556,21] := 155.191;
   DATA[2556,22] := 1.716849;
   DATA[2556,23] := 873.9682;
   DATA[2556,24] := 2.0;
   DATA[2556,25] := 2.0;
   DATA[2556,26] := 7.871251;
   DATA[2556,27] := 144.4758;
   DATA[2556,28] := 261.3753;
   DATA[2556,29] := 12.03538;
   DATA[2556,30] := 1.726096;
   DATA[2556,31] := 1.281286;
   DATA[2556,32] := 0.7352687;
   DATA[2556,33] := 0.3083624;
   DATA[2556,34] := 2.0;
   DATA[2556,35] := 250.032;
   DATA[2556,36] := 1.649953;
   DATA[2556,37] := 188.8779;
   DATA[2556,38] := 0.000128152;
   DATA[2556,39] := 1.0;
   DATA[2556,40] := 1.0;
   DATA[2557,0] := 2.632034;
   DATA[2557,1] := 868.3495;
   DATA[2557,2] := 2.0;
   DATA[2557,3] := 2.0;
   DATA[2557,4] := 262.3366;
   DATA[2557,5] := 8.393873;
   DATA[2557,6] := 329.454;
   DATA[2557,7] := 2.454362;
   DATA[2557,8] := 2.0;
   DATA[2557,9] := 2.0;
   DATA[2557,10] := 2.0;
   DATA[2557,11] := 19.70997;
   DATA[2557,12] := 2.209397;
   DATA[2557,13] := 826.7512;
   DATA[2557,14] := 1.0;
   DATA[2557,15] := 2.0;
   DATA[2557,16] := 1.0;
   DATA[2557,17] := 1.0;
   DATA[2557,18] := 1.0;
   DATA[2557,19] := 2.0;
   DATA[2557,20] := 148.808;
   DATA[2557,21] := 155.191;
   DATA[2557,22] := 1.716849;
   DATA[2557,23] := 874.545;
   DATA[2557,24] := 2.0;
   DATA[2557,25] := 2.0;
   DATA[2557,26] := 7.871251;
   DATA[2557,27] := 144.4758;
   DATA[2557,28] := 261.3753;
   DATA[2557,29] := 12.03538;
   DATA[2557,30] := 1.725968;
   DATA[2557,31] := 1.272576;
   DATA[2557,32] := 0.7352687;
   DATA[2557,33] := 0.3074656;
   DATA[2557,34] := 2.0;
   DATA[2557,35] := 250.032;
   DATA[2557,36] := 1.649953;
   DATA[2557,37] := 188.8779;
   DATA[2557,38] := 0.000128152;
   DATA[2557,39] := 1.0;
   DATA[2557,40] := 1.0;
   DATA[2558,0] := 2.654453;
   DATA[2558,1] := 867.957;
   DATA[2558,2] := 2.0;
   DATA[2558,3] := 2.0;
   DATA[2558,4] := 262.3366;
   DATA[2558,5] := 8.393873;
   DATA[2558,6] := 329.454;
   DATA[2558,7] := 2.454362;
   DATA[2558,8] := 2.0;
   DATA[2558,9] := 2.0;
   DATA[2558,10] := 2.0;
   DATA[2558,11] := 19.75479;
   DATA[2558,12] := 2.209013;
   DATA[2558,13] := 827.0716;
   DATA[2558,14] := 1.0;
   DATA[2558,15] := 2.0;
   DATA[2558,16] := 1.0;
   DATA[2558,17] := 1.0;
   DATA[2558,18] := 1.0;
   DATA[2558,19] := 2.0;
   DATA[2558,20] := 148.808;
   DATA[2558,21] := 155.191;
   DATA[2558,22] := 1.715952;
   DATA[2558,23] := 874.6988;
   DATA[2558,24] := 2.0;
   DATA[2558,25] := 2.0;
   DATA[2558,26] := 7.872533;
   DATA[2558,27] := 144.4758;
   DATA[2558,28] := 261.3753;
   DATA[2558,29] := 12.03538;
   DATA[2558,30] := 1.725968;
   DATA[2558,31] := 1.271935;
   DATA[2558,32] := 0.7352687;
   DATA[2558,33] := 0.3081703;
   DATA[2558,34] := 2.0;
   DATA[2558,35] := 250.032;
   DATA[2558,36] := 1.649953;
   DATA[2558,37] := 188.8779;
   DATA[2558,38] := 0.000128152;
   DATA[2558,39] := 1.0;
   DATA[2558,40] := 1.0;
   DATA[2559,0] := 2.670788;
   DATA[2559,1] := 867.957;
   DATA[2559,2] := 2.0;
   DATA[2559,3] := 2.0;
   DATA[2559,4] := 262.3366;
   DATA[2559,5] := 8.393873;
   DATA[2559,6] := 329.454;
   DATA[2559,7] := 2.454362;
   DATA[2559,8] := 2.0;
   DATA[2559,9] := 2.0;
   DATA[2559,10] := 2.0;
   DATA[2559,11] := 19.76759;
   DATA[2559,12] := 2.209013;
   DATA[2559,13] := 827.0316;
   DATA[2559,14] := 1.0;
   DATA[2559,15] := 2.0;
   DATA[2559,16] := 1.0;
   DATA[2559,17] := 1.0;
   DATA[2559,18] := 1.0;
   DATA[2559,19] := 2.0;
   DATA[2559,20] := 148.808;
   DATA[2559,21] := 155.191;
   DATA[2559,22] := 1.715952;
   DATA[2559,23] := 874.4296;
   DATA[2559,24] := 2.0;
   DATA[2559,25] := 2.0;
   DATA[2559,26] := 7.873174;
   DATA[2559,27] := 144.4758;
   DATA[2559,28] := 261.3753;
   DATA[2559,29] := 12.03538;
   DATA[2559,30] := 1.725968;
   DATA[2559,31] := 1.263097;
   DATA[2559,32] := 0.7352687;
   DATA[2559,33] := 0.3086827;
   DATA[2559,34] := 2.0;
   DATA[2559,35] := 250.032;
   DATA[2559,36] := 1.649953;
   DATA[2559,37] := 188.8779;
   DATA[2559,38] := 0.000128152;
   DATA[2559,39] := 1.0;
   DATA[2559,40] := 1.0;
   DATA[2560,0] := 2.670788;
   DATA[2560,1] := 868.1533;
   DATA[2560,2] := 2.0;
   DATA[2560,3] := 2.0;
   DATA[2560,4] := 262.3366;
   DATA[2560,5] := 8.393873;
   DATA[2560,6] := 329.454;
   DATA[2560,7] := 2.454362;
   DATA[2560,8] := 2.0;
   DATA[2560,9] := 2.0;
   DATA[2560,10] := 2.0;
   DATA[2560,11] := 19.81241;
   DATA[2560,12] := 2.209013;
   DATA[2560,13] := 827.1918;
   DATA[2560,14] := 1.0;
   DATA[2560,15] := 2.0;
   DATA[2560,16] := 1.0;
   DATA[2560,17] := 1.0;
   DATA[2560,18] := 1.0;
   DATA[2560,19] := 2.0;
   DATA[2560,20] := 148.808;
   DATA[2560,21] := 155.191;
   DATA[2560,22] := 1.715952;
   DATA[2560,23] := 874.3912;
   DATA[2560,24] := 2.0;
   DATA[2560,25] := 2.0;
   DATA[2560,26] := 7.873174;
   DATA[2560,27] := 144.4758;
   DATA[2560,28] := 261.3753;
   DATA[2560,29] := 12.03538;
   DATA[2560,30] := 1.725968;
   DATA[2560,31] := 1.261304;
   DATA[2560,32] := 0.7352687;
   DATA[2560,33] := 0.3086827;
   DATA[2560,34] := 2.0;
   DATA[2560,35] := 250.032;
   DATA[2560,36] := 1.649953;
   DATA[2560,37] := 188.8779;
   DATA[2560,38] := 0.000128152;
   DATA[2560,39] := 1.0;
   DATA[2560,40] := 1.0;
   DATA[2561,0] := 2.652532;
   DATA[2561,1] := 867.6822;
   DATA[2561,2] := 2.0;
   DATA[2561,3] := 2.0;
   DATA[2561,4] := 262.3366;
   DATA[2561,5] := 8.393873;
   DATA[2561,6] := 329.454;
   DATA[2561,7] := 2.455515;
   DATA[2561,8] := 2.0;
   DATA[2561,9] := 2.0;
   DATA[2561,10] := 2.0;
   DATA[2561,11] := 19.81241;
   DATA[2561,12] := 2.209013;
   DATA[2561,13] := 827.2719;
   DATA[2561,14] := 1.0;
   DATA[2561,15] := 2.0;
   DATA[2561,16] := 1.0;
   DATA[2561,17] := 1.0;
   DATA[2561,18] := 1.0;
   DATA[2561,19] := 2.0;
   DATA[2561,20] := 148.808;
   DATA[2561,21] := 155.191;
   DATA[2561,22] := 1.715952;
   DATA[2561,23] := 874.6988;
   DATA[2561,24] := 2.0;
   DATA[2561,25] := 2.0;
   DATA[2561,26] := 7.873174;
   DATA[2561,27] := 144.4758;
   DATA[2561,28] := 261.3753;
   DATA[2561,29] := 12.03538;
   DATA[2561,30] := 1.726865;
   DATA[2561,31] := 1.261304;
   DATA[2561,32] := 0.7352687;
   DATA[2561,33] := 0.3086827;
   DATA[2561,34] := 2.0;
   DATA[2561,35] := 250.032;
   DATA[2561,36] := 1.649953;
   DATA[2561,37] := 188.8779;
   DATA[2561,38] := 0.000128152;
   DATA[2561,39] := 1.0;
   DATA[2561,40] := 1.0;
   DATA[2562,0] := 2.628191;
   DATA[2562,1] := 867.2897;
   DATA[2562,2] := 2.0;
   DATA[2562,3] := 2.0;
   DATA[2562,4] := 262.3366;
   DATA[2562,5] := 8.393873;
   DATA[2562,6] := 329.454;
   DATA[2562,7] := 2.456541;
   DATA[2562,8] := 2.0;
   DATA[2562,9] := 2.0;
   DATA[2562,10] := 2.0;
   DATA[2562,11] := 19.81241;
   DATA[2562,12] := 2.209397;
   DATA[2562,13] := 827.1918;
   DATA[2562,14] := 1.0;
   DATA[2562,15] := 2.0;
   DATA[2562,16] := 1.0;
   DATA[2562,17] := 1.0;
   DATA[2562,18] := 1.0;
   DATA[2562,19] := 2.0;
   DATA[2562,20] := 148.808;
   DATA[2562,21] := 155.191;
   DATA[2562,22] := 1.715952;
   DATA[2562,23] := 874.545;
   DATA[2562,24] := 2.0;
   DATA[2562,25] := 2.0;
   DATA[2562,26] := 7.873174;
   DATA[2562,27] := 144.4758;
   DATA[2562,28] := 261.3753;
   DATA[2562,29] := 12.03538;
   DATA[2562,30] := 1.726865;
   DATA[2562,31] := 1.280646;
   DATA[2562,32] := 0.7352687;
   DATA[2562,33] := 0.3086827;
   DATA[2562,34] := 2.0;
   DATA[2562,35] := 250.0801;
   DATA[2562,36] := 1.649953;
   DATA[2562,37] := 188.8779;
   DATA[2562,38] := 0.000128152;
   DATA[2562,39] := 1.0;
   DATA[2562,40] := 1.0;
   DATA[2563,0] := 2.620184;
   DATA[2563,1] := 867.3289;
   DATA[2563,2] := 2.0;
   DATA[2563,3] := 2.0;
   DATA[2563,4] := 262.3366;
   DATA[2563,5] := 8.393873;
   DATA[2563,6] := 329.454;
   DATA[2563,7] := 2.456541;
   DATA[2563,8] := 2.0;
   DATA[2563,9] := 2.0;
   DATA[2563,10] := 2.0;
   DATA[2563,11] := 19.81241;
   DATA[2563,12] := 2.209525;
   DATA[2563,13] := 827.352;
   DATA[2563,14] := 1.0;
   DATA[2563,15] := 2.0;
   DATA[2563,16] := 1.0;
   DATA[2563,17] := 1.0;
   DATA[2563,18] := 1.0;
   DATA[2563,19] := 2.0;
   DATA[2563,20] := 148.808;
   DATA[2563,21] := 155.191;
   DATA[2563,22] := 1.717746;
   DATA[2563,23] := 874.3527;
   DATA[2563,24] := 2.0;
   DATA[2563,25] := 2.0;
   DATA[2563,26] := 7.873174;
   DATA[2563,27] := 144.4758;
   DATA[2563,28] := 261.3753;
   DATA[2563,29] := 12.03538;
   DATA[2563,30] := 1.726865;
   DATA[2563,31] := 1.281542;
   DATA[2563,32] := 0.7352687;
   DATA[2563,33] := 0.3084265;
   DATA[2563,34] := 2.0;
   DATA[2563,35] := 250.1923;
   DATA[2563,36] := 1.649953;
   DATA[2563,37] := 188.8779;
   DATA[2563,38] := 0.000128152;
   DATA[2563,39] := 1.0;
   DATA[2563,40] := 1.0;
   DATA[2564,0] := 2.610575;
   DATA[2564,1] := 867.0934;
   DATA[2564,2] := 2.0;
   DATA[2564,3] := 2.0;
   DATA[2564,4] := 262.3366;
   DATA[2564,5] := 8.393873;
   DATA[2564,6] := 329.454;
   DATA[2564,7] := 2.454618;
   DATA[2564,8] := 2.0;
   DATA[2564,9] := 2.0;
   DATA[2564,10] := 2.0;
   DATA[2564,11] := 19.81241;
   DATA[2564,12] := 2.210037;
   DATA[2564,13] := 827.2318;
   DATA[2564,14] := 1.0;
   DATA[2564,15] := 2.0;
   DATA[2564,16] := 1.0;
   DATA[2564,17] := 1.0;
   DATA[2564,18] := 1.0;
   DATA[2564,19] := 2.0;
   DATA[2564,20] := 148.808;
   DATA[2564,21] := 155.191;
   DATA[2564,22] := 1.719284;
   DATA[2564,23] := 874.5065;
   DATA[2564,24] := 2.0;
   DATA[2564,25] := 2.0;
   DATA[2564,26] := 7.873174;
   DATA[2564,27] := 144.4758;
   DATA[2564,28] := 261.3753;
   DATA[2564,29] := 12.03538;
   DATA[2564,30] := 1.726865;
   DATA[2564,31] := 1.282183;
   DATA[2564,32] := 0.7352687;
   DATA[2564,33] := 0.3083624;
   DATA[2564,34] := 2.0;
   DATA[2564,35] := 250.1923;
   DATA[2564,36] := 1.649953;
   DATA[2564,37] := 188.8779;
   DATA[2564,38] := 0.000128152;
   DATA[2564,39] := 1.0;
   DATA[2564,40] := 1.0;
   DATA[2565,0] := 2.585914;
   DATA[2565,1] := 867.0542;
   DATA[2565,2] := 2.0;
   DATA[2565,3] := 2.0;
   DATA[2565,4] := 262.3366;
   DATA[2565,5] := 8.393873;
   DATA[2565,6] := 329.454;
   DATA[2565,7] := 2.453209;
   DATA[2565,8] := 2.0;
   DATA[2565,9] := 2.0;
   DATA[2565,10] := 2.0;
   DATA[2565,11] := 19.69076;
   DATA[2565,12] := 2.21055;
   DATA[2565,13] := 827.1517;
   DATA[2565,14] := 1.0;
   DATA[2565,15] := 2.0;
   DATA[2565,16] := 1.0;
   DATA[2565,17] := 1.0;
   DATA[2565,18] := 1.0;
   DATA[2565,19] := 2.0;
   DATA[2565,20] := 148.808;
   DATA[2565,21] := 155.191;
   DATA[2565,22] := 1.719284;
   DATA[2565,23] := 874.6219;
   DATA[2565,24] := 2.0;
   DATA[2565,25] := 2.0;
   DATA[2565,26] := 7.873174;
   DATA[2565,27] := 144.4758;
   DATA[2565,28] := 261.3753;
   DATA[2565,29] := 12.03538;
   DATA[2565,30] := 1.726865;
   DATA[2565,31] := 1.289868;
   DATA[2565,32] := 0.7352687;
   DATA[2565,33] := 0.3072094;
   DATA[2565,34] := 2.0;
   DATA[2565,35] := 250.1923;
   DATA[2565,36] := 1.730048;
   DATA[2565,37] := 188.8779;
   DATA[2565,38] := 0.000128152;
   DATA[2565,39] := 1.0;
   DATA[2565,40] := 1.0;
   DATA[2566,0] := 2.561573;
   DATA[2566,1] := 867.0934;
   DATA[2566,2] := 2.0;
   DATA[2566,3] := 2.0;
   DATA[2566,4] := 262.3366;
   DATA[2566,5] := 8.393873;
   DATA[2566,6] := 329.454;
   DATA[2566,7] := 2.453209;
   DATA[2566,8] := 2.0;
   DATA[2566,9] := 2.0;
   DATA[2566,10] := 2.0;
   DATA[2566,11] := 19.67796;
   DATA[2566,12] := 2.21055;
   DATA[2566,13] := 827.0716;
   DATA[2566,14] := 1.0;
   DATA[2566,15] := 2.0;
   DATA[2566,16] := 1.0;
   DATA[2566,17] := 1.0;
   DATA[2566,18] := 1.0;
   DATA[2566,19] := 2.0;
   DATA[2566,20] := 148.808;
   DATA[2566,21] := 155.191;
   DATA[2566,22] := 1.719284;
   DATA[2566,23] := 874.3912;
   DATA[2566,24] := 2.0;
   DATA[2566,25] := 2.0;
   DATA[2566,26] := 7.874135;
   DATA[2566,27] := 144.4758;
   DATA[2566,28] := 261.3753;
   DATA[2566,29] := 12.03538;
   DATA[2566,30] := 1.726865;
   DATA[2566,31] := 1.290509;
   DATA[2566,32] := 0.7352687;
   DATA[2566,33] := 0.306761;
   DATA[2566,34] := 2.0;
   DATA[2566,35] := 250.1923;
   DATA[2566,36] := 1.730048;
   DATA[2566,37] := 188.8779;
   DATA[2566,38] := 0.000128152;
   DATA[2566,39] := 1.0;
   DATA[2566,40] := 1.0;
   DATA[2567,0] := 2.543958;
   DATA[2567,1] := 866.9364;
   DATA[2567,2] := 2.0;
   DATA[2567,3] := 2.0;
   DATA[2567,4] := 262.3366;
   DATA[2567,5] := 8.393873;
   DATA[2567,6] := 329.454;
   DATA[2567,7] := 2.453209;
   DATA[2567,8] := 2.0;
   DATA[2567,9] := 2.0;
   DATA[2567,10] := 2.0;
   DATA[2567,11] := 19.66835;
   DATA[2567,12] := 2.209269;
   DATA[2567,13] := 827.352;
   DATA[2567,14] := 1.0;
   DATA[2567,15] := 2.0;
   DATA[2567,16] := 1.0;
   DATA[2567,17] := 1.0;
   DATA[2567,18] := 1.0;
   DATA[2567,19] := 2.0;
   DATA[2567,20] := 148.808;
   DATA[2567,21] := 155.191;
   DATA[2567,22] := 1.719284;
   DATA[2567,23] := 874.0451;
   DATA[2567,24] := 2.0;
   DATA[2567,25] := 2.0;
   DATA[2567,26] := 7.874776;
   DATA[2567,27] := 144.4758;
   DATA[2567,28] := 261.3753;
   DATA[2567,29] := 12.03538;
   DATA[2567,30] := 1.726865;
   DATA[2567,31] := 1.27296;
   DATA[2567,32] := 0.7352687;
   DATA[2567,33] := 0.3064407;
   DATA[2567,34] := 2.0;
   DATA[2567,35] := 250.1923;
   DATA[2567,36] := 1.730048;
   DATA[2567,37] := 188.8779;
   DATA[2567,38] := 0.000128152;
   DATA[2567,39] := 1.0;
   DATA[2567,40] := 1.0;
   DATA[2568,0] := 2.526022;
   DATA[2568,1] := 867.3682;
   DATA[2568,2] := 2.0;
   DATA[2568,3] := 2.0;
   DATA[2568,4] := 262.3366;
   DATA[2568,5] := 8.393873;
   DATA[2568,6] := 329.454;
   DATA[2568,7] := 2.453209;
   DATA[2568,8] := 2.0;
   DATA[2568,9] := 2.0;
   DATA[2568,10] := 2.0;
   DATA[2568,11] := 19.66835;
   DATA[2568,12] := 2.206322;
   DATA[2568,13] := 827.2719;
   DATA[2568,14] := 1.0;
   DATA[2568,15] := 2.0;
   DATA[2568,16] := 1.0;
   DATA[2568,17] := 1.0;
   DATA[2568,18] := 1.0;
   DATA[2568,19] := 2.0;
   DATA[2568,20] := 148.808;
   DATA[2568,21] := 155.191;
   DATA[2568,22] := 1.719284;
   DATA[2568,23] := 874.122;
   DATA[2568,24] := 2.0;
   DATA[2568,25] := 2.0;
   DATA[2568,26] := 7.874776;
   DATA[2568,27] := 144.4758;
   DATA[2568,28] := 261.3753;
   DATA[2568,29] := 12.03538;
   DATA[2568,30] := 1.726865;
   DATA[2568,31] := 1.272704;
   DATA[2568,32] := 0.7352687;
   DATA[2568,33] := 0.3081062;
   DATA[2568,34] := 2.0;
   DATA[2568,35] := 250.0961;
   DATA[2568,36] := 1.730048;
   DATA[2568,37] := 188.8779;
   DATA[2568,38] := 0.000128152;
   DATA[2568,39] := 1.0;
   DATA[2568,40] := 1.0;
   DATA[2569,0] := 2.507126;
   DATA[2569,1] := 867.0934;
   DATA[2569,2] := 2.0;
   DATA[2569,3] := 2.0;
   DATA[2569,4] := 262.3366;
   DATA[2569,5] := 8.393873;
   DATA[2569,6] := 329.454;
   DATA[2569,7] := 2.45449;
   DATA[2569,8] := 2.0;
   DATA[2569,9] := 2.0;
   DATA[2569,10] := 2.0;
   DATA[2569,11] := 19.75159;
   DATA[2569,12] := 2.206322;
   DATA[2569,13] := 827.7926;
   DATA[2569,14] := 1.0;
   DATA[2569,15] := 2.0;
   DATA[2569,16] := 1.0;
   DATA[2569,17] := 1.0;
   DATA[2569,18] := 1.0;
   DATA[2569,19] := 2.0;
   DATA[2569,20] := 148.808;
   DATA[2569,21] := 155.191;
   DATA[2569,22] := 1.716592;
   DATA[2569,23] := 873.9682;
   DATA[2569,24] := 2.0;
   DATA[2569,25] := 2.0;
   DATA[2569,26] := 7.874776;
   DATA[2569,27] := 144.4758;
   DATA[2569,28] := 261.3753;
   DATA[2569,29] := 12.03538;
   DATA[2569,30] := 1.72507;
   DATA[2569,31] := 1.276419;
   DATA[2569,32] := 0.7352687;
   DATA[2569,33] := 0.3084265;
   DATA[2569,34] := 2.0;
   DATA[2569,35] := 249.9519;
   DATA[2569,36] := 1.730048;
   DATA[2569,37] := 188.8779;
   DATA[2569,38] := 0.000128152;
   DATA[2569,39] := 1.0;
   DATA[2569,40] := 1.0;
   DATA[2570,0] := 2.490472;
   DATA[2570,1] := 867.3289;
   DATA[2570,2] := 2.0;
   DATA[2570,3] := 2.0;
   DATA[2570,4] := 262.3366;
   DATA[2570,5] := 8.393873;
   DATA[2570,6] := 329.454;
   DATA[2570,7] := 2.456156;
   DATA[2570,8] := 2.0;
   DATA[2570,9] := 2.0;
   DATA[2570,10] := 2.0;
   DATA[2570,11] := 19.76439;
   DATA[2570,12] := 2.206322;
   DATA[2570,13] := 827.8326;
   DATA[2570,14] := 1.0;
   DATA[2570,15] := 2.0;
   DATA[2570,16] := 1.0;
   DATA[2570,17] := 1.0;
   DATA[2570,18] := 1.0;
   DATA[2570,19] := 2.0;
   DATA[2570,20] := 148.808;
   DATA[2570,21] := 155.0115;
   DATA[2570,22] := 1.715824;
   DATA[2570,23] := 873.7375;
   DATA[2570,24] := 2.0;
   DATA[2570,25] := 2.0;
   DATA[2570,26] := 7.874776;
   DATA[2570,27] := 144.4758;
   DATA[2570,28] := 261.3753;
   DATA[2570,29] := 12.03538;
   DATA[2570,30] := 1.724814;
   DATA[2570,31] := 1.272064;
   DATA[2570,32] := 0.7352687;
   DATA[2570,33] := 0.3084265;
   DATA[2570,34] := 2.0;
   DATA[2570,35] := 249.7597;
   DATA[2570,36] := 1.730048;
   DATA[2570,37] := 188.8779;
   DATA[2570,38] := 0.000128152;
   DATA[2570,39] := 1.0;
   DATA[2570,40] := 1.0;
   DATA[2571,0] := 2.470294;
   DATA[2571,1] := 867.486;
   DATA[2571,2] := 2.0;
   DATA[2571,3] := 2.0;
   DATA[2571,4] := 262.3366;
   DATA[2571,5] := 8.393873;
   DATA[2571,6] := 329.454;
   DATA[2571,7] := 2.456156;
   DATA[2571,8] := 2.0;
   DATA[2571,9] := 2.0;
   DATA[2571,10] := 2.0;
   DATA[2571,11] := 19.77079;
   DATA[2571,12] := 2.206322;
   DATA[2571,13] := 827.9929;
   DATA[2571,14] := 1.0;
   DATA[2571,15] := 2.0;
   DATA[2571,16] := 1.0;
   DATA[2571,17] := 1.0;
   DATA[2571,18] := 1.0;
   DATA[2571,19] := 2.0;
   DATA[2571,20] := 148.808;
   DATA[2571,21] := 155.0115;
   DATA[2571,22] := 1.715824;
   DATA[2571,23] := 873.8144;
   DATA[2571,24] := 2.0;
   DATA[2571,25] := 2.0;
   DATA[2571,26] := 7.874776;
   DATA[2571,27] := 144.4758;
   DATA[2571,28] := 261.3753;
   DATA[2571,29] := 12.03538;
   DATA[2571,30] := 1.724814;
   DATA[2571,31] := 1.291277;
   DATA[2571,32] := 0.7352687;
   DATA[2571,33] := 0.3084265;
   DATA[2571,34] := 2.0;
   DATA[2571,35] := 249.7437;
   DATA[2571,36] := 1.730048;
   DATA[2571,37] := 188.6375;
   DATA[2571,38] := 0.000128152;
   DATA[2571,39] := 1.0;
   DATA[2571,40] := 1.0;
   DATA[2572,0] := 2.452679;
   DATA[2572,1] := 867.486;
   DATA[2572,2] := 2.0;
   DATA[2572,3] := 2.0;
   DATA[2572,4] := 262.3366;
   DATA[2572,5] := 8.393873;
   DATA[2572,6] := 329.454;
   DATA[2572,7] := 2.456156;
   DATA[2572,8] := 2.0;
   DATA[2572,9] := 2.0;
   DATA[2572,10] := 2.0;
   DATA[2572,11] := 19.77079;
   DATA[2572,12] := 2.208628;
   DATA[2572,13] := 828.3533;
   DATA[2572,14] := 1.0;
   DATA[2572,15] := 2.0;
   DATA[2572,16] := 1.0;
   DATA[2572,17] := 1.0;
   DATA[2572,18] := 1.0;
   DATA[2572,19] := 2.0;
   DATA[2572,20] := 148.808;
   DATA[2572,21] := 155.0115;
   DATA[2572,22] := 1.713645;
   DATA[2572,23] := 873.7375;
   DATA[2572,24] := 2.0;
   DATA[2572,25] := 2.0;
   DATA[2572,26] := 7.874776;
   DATA[2572,27] := 144.4758;
   DATA[2572,28] := 261.3753;
   DATA[2572,29] := 12.03538;
   DATA[2572,30] := 1.724814;
   DATA[2572,31] := 1.289228;
   DATA[2572,32] := 0.7352687;
   DATA[2572,33] := 0.3084265;
   DATA[2572,34] := 2.0;
   DATA[2572,35] := 249.7437;
   DATA[2572,36] := 1.730048;
   DATA[2572,37] := 188.6375;
   DATA[2572,38] := 0.000128152;
   DATA[2572,39] := 1.0;
   DATA[2572,40] := 1.0;
   DATA[2573,0] := 2.431861;
   DATA[2573,1] := 868.2318;
   DATA[2573,2] := 2.0;
   DATA[2573,3] := 2.0;
   DATA[2573,4] := 262.3366;
   DATA[2573,5] := 8.393873;
   DATA[2573,6] := 329.4027;
   DATA[2573,7] := 2.456541;
   DATA[2573,8] := 2.0;
   DATA[2573,9] := 2.0;
   DATA[2573,10] := 2.0;
   DATA[2573,11] := 19.77079;
   DATA[2573,12] := 2.208628;
   DATA[2573,13] := 828.0729;
   DATA[2573,14] := 1.0;
   DATA[2573,15] := 2.0;
   DATA[2573,16] := 1.0;
   DATA[2573,17] := 1.0;
   DATA[2573,18] := 1.0;
   DATA[2573,19] := 2.0;
   DATA[2573,20] := 148.808;
   DATA[2573,21] := 155.191;
   DATA[2573,22] := 1.713261;
   DATA[2573,23] := 873.9297;
   DATA[2573,24] := 2.0;
   DATA[2573,25] := 2.0;
   DATA[2573,26] := 7.874776;
   DATA[2573,27] := 144.4758;
   DATA[2573,28] := 261.3753;
   DATA[2573,29] := 12.03538;
   DATA[2573,30] := 1.724814;
   DATA[2573,31] := 1.282183;
   DATA[2573,32] := 0.7352687;
   DATA[2573,33] := 0.3084265;
   DATA[2573,34] := 2.0;
   DATA[2573,35] := 249.7437;
   DATA[2573,36] := 1.649953;
   DATA[2573,37] := 188.6375;
   DATA[2573,38] := 0.000128152;
   DATA[2573,39] := 1.0;
   DATA[2573,40] := 1.0;
   DATA[2574,0] := 2.428979;
   DATA[2574,1] := 868.428;
   DATA[2574,2] := 2.0;
   DATA[2574,3] := 2.0;
   DATA[2574,4] := 262.3366;
   DATA[2574,5] := 8.393873;
   DATA[2574,6] := 329.4027;
   DATA[2574,7] := 2.456541;
   DATA[2574,8] := 2.0;
   DATA[2574,9] := 2.0;
   DATA[2574,10] := 2.0;
   DATA[2574,11] := 19.68756;
   DATA[2574,12] := 2.208628;
   DATA[2574,13] := 828.3934;
   DATA[2574,14] := 1.0;
   DATA[2574,15] := 2.0;
   DATA[2574,16] := 1.0;
   DATA[2574,17] := 1.0;
   DATA[2574,18] := 1.0;
   DATA[2574,19] := 2.0;
   DATA[2574,20] := 148.808;
   DATA[2574,21] := 155.191;
   DATA[2574,22] := 1.713261;
   DATA[2574,23] := 873.9682;
   DATA[2574,24] := 2.0;
   DATA[2574,25] := 2.0;
   DATA[2574,26] := 7.871251;
   DATA[2574,27] := 144.4758;
   DATA[2574,28] := 261.3753;
   DATA[2574,29] := 12.03538;
   DATA[2574,30] := 1.724814;
   DATA[2574,31] := 1.272576;
   DATA[2574,32] := 0.7352687;
   DATA[2574,33] := 0.3084265;
   DATA[2574,34] := 2.0;
   DATA[2574,35] := 249.6155;
   DATA[2574,36] := 1.649953;
   DATA[2574,37] := 188.5254;
   DATA[2574,38] := 0.000128152;
   DATA[2574,39] := 1.0;
   DATA[2574,40] := 1.0;
   DATA[2575,0] := 2.428018;
   DATA[2575,1] := 868.4673;
   DATA[2575,2] := 2.0;
   DATA[2575,3] := 2.0;
   DATA[2575,4] := 262.3366;
   DATA[2575,5] := 8.393873;
   DATA[2575,6] := 329.4027;
   DATA[2575,7] := 2.453209;
   DATA[2575,8] := 2.0;
   DATA[2575,9] := 2.0;
   DATA[2575,10] := 2.0;
   DATA[2575,11] := 19.68756;
   DATA[2575,12] := 2.208628;
   DATA[2575,13] := 828.5936;
   DATA[2575,14] := 1.0;
   DATA[2575,15] := 2.0;
   DATA[2575,16] := 1.0;
   DATA[2575,17] := 1.0;
   DATA[2575,18] := 1.0;
   DATA[2575,19] := 2.0;
   DATA[2575,20] := 148.808;
   DATA[2575,21] := 155.191;
   DATA[2575,22] := 1.713261;
   DATA[2575,23] := 874.2374;
   DATA[2575,24] := 2.0;
   DATA[2575,25] := 2.0;
   DATA[2575,26] := 7.871251;
   DATA[2575,27] := 144.4758;
   DATA[2575,28] := 261.3753;
   DATA[2575,29] := 12.03538;
   DATA[2575,30] := 1.724301;
   DATA[2575,31] := 1.275266;
   DATA[2575,32] := 0.7352687;
   DATA[2575,33] := 0.3084265;
   DATA[2575,34] := 2.0;
   DATA[2575,35] := 249.6155;
   DATA[2575,36] := 1.649953;
   DATA[2575,37] := 188.5254;
   DATA[2575,38] := 0.000128152;
   DATA[2575,39] := 1.0;
   DATA[2575,40] := 1.0;
   DATA[2576,0] := 2.452359;
   DATA[2576,1] := 868.4673;
   DATA[2576,2] := 2.0;
   DATA[2576,3] := 2.0;
   DATA[2576,4] := 262.3366;
   DATA[2576,5] := 8.394835;
   DATA[2576,6] := 329.4027;
   DATA[2576,7] := 2.452312;
   DATA[2576,8] := 2.0;
   DATA[2576,9] := 2.0;
   DATA[2576,10] := 2.0;
   DATA[2576,11] := 19.68756;
   DATA[2576,12] := 2.208628;
   DATA[2576,13] := 828.3934;
   DATA[2576,14] := 1.0;
   DATA[2576,15] := 2.0;
   DATA[2576,16] := 1.0;
   DATA[2576,17] := 1.0;
   DATA[2576,18] := 1.0;
   DATA[2576,19] := 2.0;
   DATA[2576,20] := 148.808;
   DATA[2576,21] := 155.191;
   DATA[2576,22] := 1.713261;
   DATA[2576,23] := 874.5065;
   DATA[2576,24] := 2.0;
   DATA[2576,25] := 2.0;
   DATA[2576,26] := 7.871251;
   DATA[2576,27] := 144.4758;
   DATA[2576,28] := 261.3753;
   DATA[2576,29] := 12.03538;
   DATA[2576,30] := 1.724301;
   DATA[2576,31] := 1.280902;
   DATA[2576,32] := 0.7352687;
   DATA[2576,33] := 0.3084265;
   DATA[2576,34] := 2.0;
   DATA[2576,35] := 249.6155;
   DATA[2576,36] := 1.649953;
   DATA[2576,37] := 188.5254;
   DATA[2576,38] := 0.000128152;
   DATA[2576,39] := 1.0;
   DATA[2576,40] := 1.0;
   DATA[2577,0] := 2.503283;
   DATA[2577,1] := 868.7421;
   DATA[2577,2] := 2.0;
   DATA[2577,3] := 2.0;
   DATA[2577,4] := 262.3366;
   DATA[2577,5] := 8.396437;
   DATA[2577,6] := 329.4027;
   DATA[2577,7] := 2.452312;
   DATA[2577,8] := 2.0;
   DATA[2577,9] := 2.0;
   DATA[2577,10] := 2.0;
   DATA[2577,11] := 19.68756;
   DATA[2577,12] := 2.208628;
